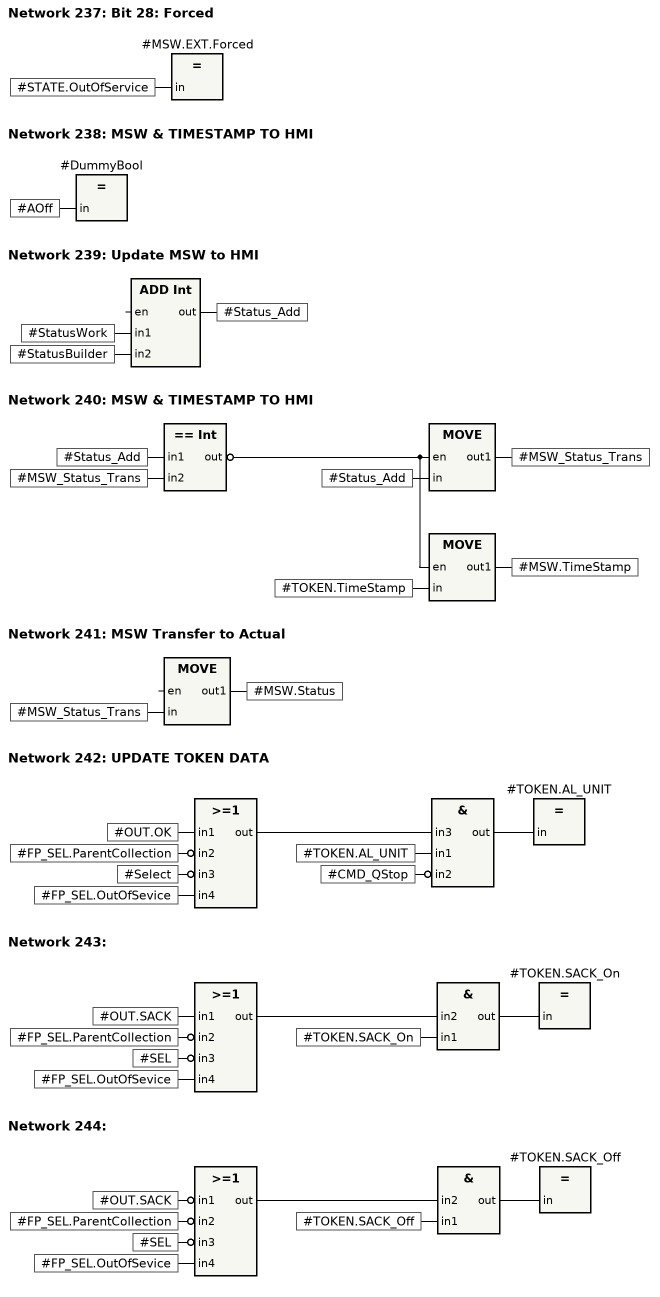
   #MSW.EXT.Forced := #STATE.OutOfService;
END_REGION

REGION Network 238: MSW & TIMESTAMP TO HMI
   #DummyBool := #AOff;
END_REGION

REGION Network 239: Update MSW to HMI
   #Status_Add := #StatusWork + #StatusBuilder;
END_REGION

REGION Network 240: MSW & TIMESTAMP TO HMI
   #_w1 := NOT (#Status_Add = #MSW_Status_Trans);
   IF #_w1 THEN
       #MSW_Status_Trans := #Status_Add;
       #MSW.TimeStamp := #TOKEN.TimeStamp;
   END_IF;
END_REGION

REGION Network 241: MSW Transfer to Actual
   #MSW.Status := #MSW_Status_Trans;
END_REGION

REGION Network 242: UPDATE TOKEN DATA
   #TOKEN.AL_UNIT := (#OUT.OK OR NOT #FP_SEL.ParentCollection OR NOT #Select OR #FP_SEL.OutOfSevice) AND #TOKEN.AL_UNIT AND NOT #CMD_QStop;
END_REGION

REGION Network 243
   // Build 005 - 24.June.2020 (MIA-US): Replace "Select" with "SEL"
   #TOKEN.SACK_On := (#OUT.SACK OR NOT #FP_SEL.ParentCollection OR NOT #SEL OR #FP_SEL.OutOfSevice) AND #TOKEN.SACK_On;
END_REGION

REGION Network 244
   #TOKEN.SACK_Off := (NOT #OUT.SACK OR NOT #FP_SEL.ParentCollection OR NOT #SEL OR #FP_SEL.OutOfSevice) AND #TOKEN.SACK_Off;
END_REGION

REGION Network 245
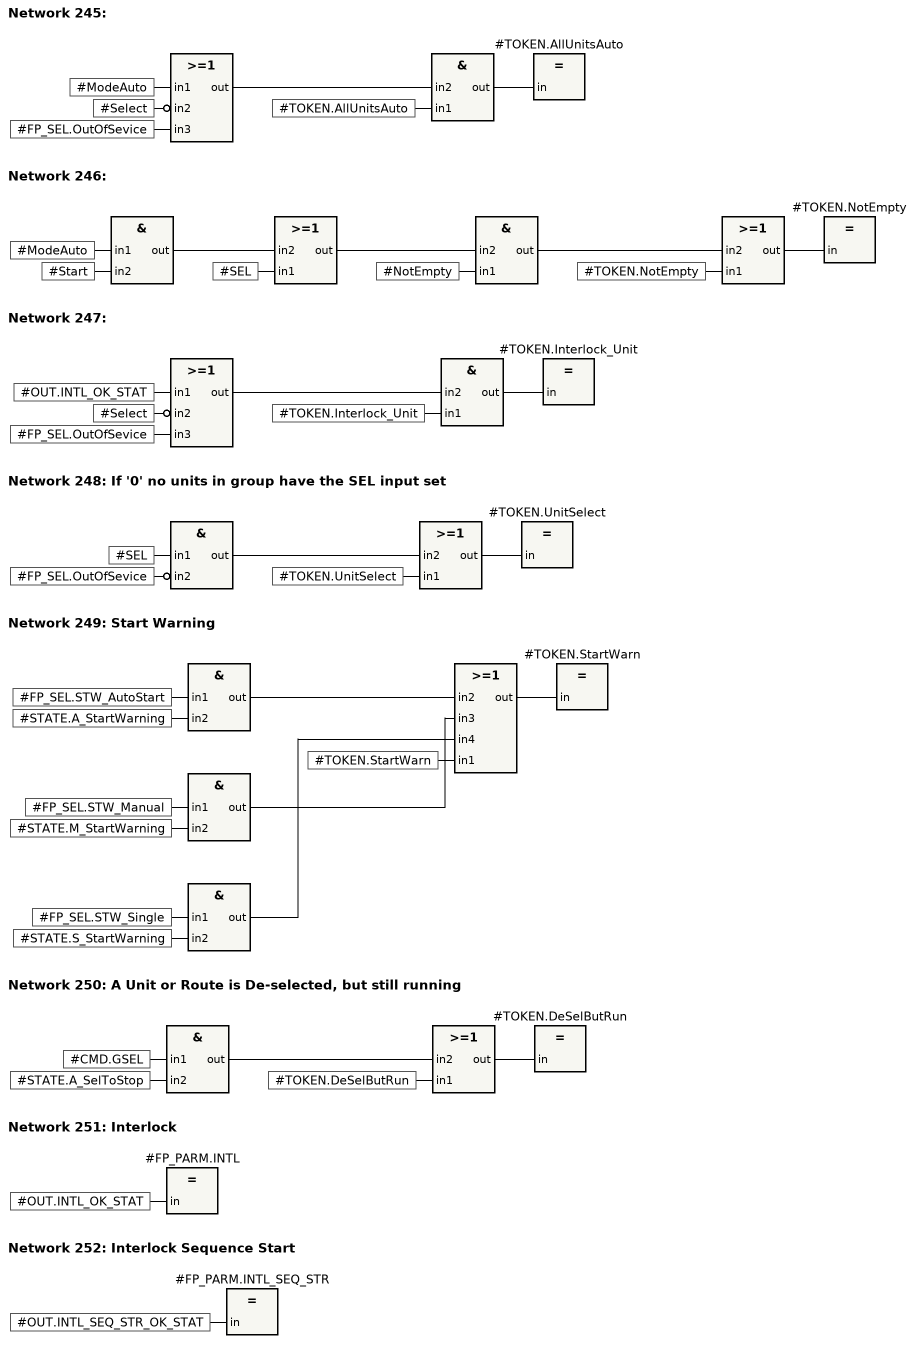
   #TOKEN.AllUnitsAuto := (#ModeAuto OR NOT #Select OR #FP_SEL.OutOfSevice) AND #TOKEN.AllUnitsAuto;
END_REGION

REGION Network 246
   #TOKEN.NotEmpty := (((#ModeAuto AND #Start) OR #SEL) AND #NotEmpty) OR #TOKEN.NotEmpty;
END_REGION

REGION Network 247
   #TOKEN.Interlock_Unit := (#OUT.INTL_OK_STAT OR NOT #Select OR #FP_SEL.OutOfSevice) AND #TOKEN.Interlock_Unit;
END_REGION

REGION Network 248: If '0' no units in group have the SEL input set
   #TOKEN.UnitSelect := (#SEL AND NOT #FP_SEL.OutOfSevice) OR #TOKEN.UnitSelect;
END_REGION

REGION Network 249: Start Warning
   #TOKEN.StartWarn := (#FP_SEL.STW_AutoStart AND #STATE.A_StartWarning) OR (#FP_SEL.STW_Manual AND #STATE.M_StartWarning) OR (#FP_SEL.STW_Single AND #STATE.S_StartWarning) OR #TOKEN.StartWarn;
END_REGION

REGION Network 250: A Unit or Route is De-selected, but still running
   #TOKEN.DeSelButRun := (#CMD.GSEL AND #STATE.A_SelToStop) OR #TOKEN.DeSelButRun;
END_REGION

REGION Network 251: Interlock
   #FP_PARM.INTL := #OUT.INTL_OK_STAT;
END_REGION

REGION Network 252: Interlock Sequence Start
   #FP_PARM.INTL_SEQ_STR := #OUT.INTL_SEQ_STR_OK_STAT;
END_REGION

REGION Network 253: Interlock Status to HMI
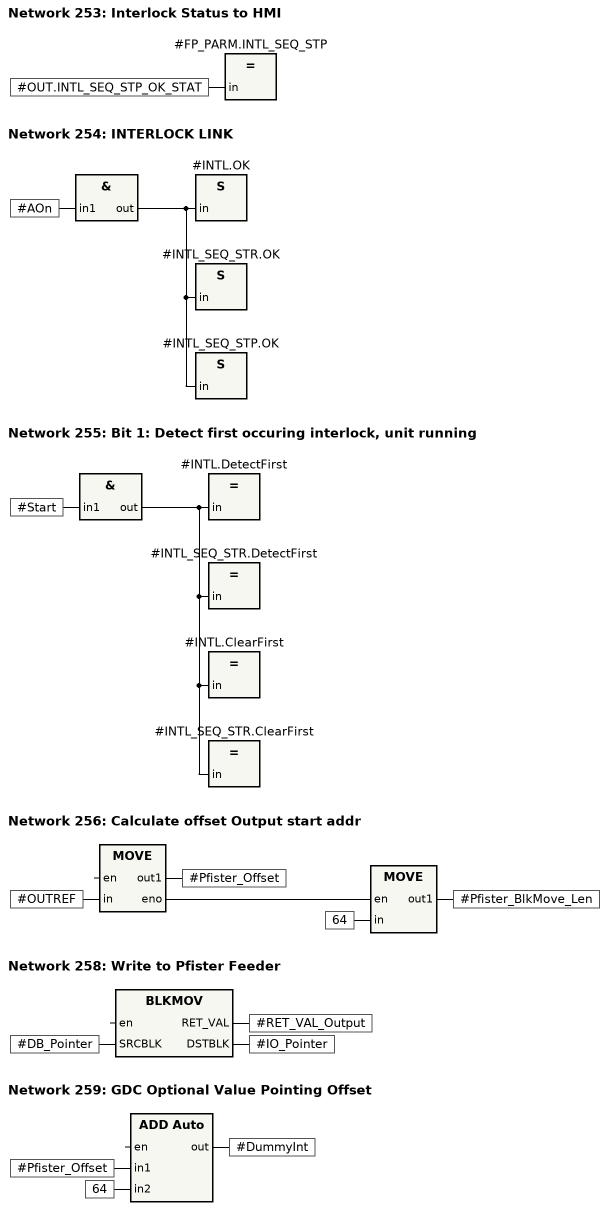
   #FP_PARM.INTL_SEQ_STP := #OUT.INTL_SEQ_STP_OK_STAT;
END_REGION

REGION Network 254: INTERLOCK LINK
   IF #AOn THEN
       #INTL.OK := TRUE;
       #INTL_SEQ_STR.OK := TRUE;
       #INTL_SEQ_STP.OK := TRUE;
   END_IF;
END_REGION

REGION Network 255: Bit 1: Detect first occuring interlock, unit running
   #INTL.DetectFirst := #Start;
   #INTL_SEQ_STR.DetectFirst := #Start;
   #INTL.ClearFirst := #Start;
   #INTL_SEQ_STR.ClearFirst := #Start;
END_REGION

REGION Network 256: Calculate offset Output start addr
   #Pfister_Offset := #OUTREF;
   #Pfister_BlkMove_Len := 64;
END_REGION

REGION Network 257 (STL): Target Pointers Sending Output Data
         LAR1;  // Make AR1 pointer to Unit Output
         L     16#10;  // ANY Syntax ID
         T     LB[AR1, P#0.0];  // ..Store Byte 0
         L     16#02;  // Data Type = Byte
         T     LB[AR1, P#1.0];  // ..Store Byte 1
         L     #Pfister_BlkMove_Len;  // Load Packed length
         T     LW[AR1, P#2.0];  // ..Store byte 2/3
         L     0;  // used with DB else "0"
         T     LW[AR1, P#4.0];  // ..Store byte 4/5
         L     #Pfister_Offset;  // Source offset (Variable for Node's)
         SLD   3;  // with offset
         OD    16#8200_0000;  // Output Area (I/O) Code (S7)
         T     LD[AR1, P#6.0];  // ..Store byte 6/7/8/9

         LAR1;  // Load start point of cyclic data
         TAR1  #DummyDWord;  // Store in temp. point
         L     #DummyDWord;  // Load temp. point
         T     #Addr_InstanceDB;  // Store start point as DB address

         LAR1;  // Make AR1 point to calling program stack
         L     16#10;  // ANY Syntax ID
         T     LB[AR1, P#0.0];  // ..Store Byte 0
         L     16#02;  // Data Type = Byte
         T     LB[AR1, P#1.0];  // ..Store Byte 1
         L     #Pfister_BlkMove_Len;  // Load Packed length
         T     LW[AR1, P#2.0];  // ..Store Byte 2/3
         L     #BlockInfo.DB_Number;  // used with DB use No. else "0"
         T     LW[AR1, P#4.0];  // ..Store byte 4/5
         L     #Addr_InstanceDB;  // Load Instance DB Start address
         L     16#8500_0000;
         -D;
         L     16#8400_0000;
         +D;
         T     LD[AR1, P#6.0];  // ..Store byte 6/7/8/9
END_REGION

REGION Network 258: Write to Pfister Feeder
   #RET_VAL_Output := BLKMOV(SRCBLK := #DB_Pointer, DSTBLK => #IO_Pointer);
END_REGION

REGION Network 259: GDC Optional Value Pointing Offset
   // Build 07 - 09 Jan 2022(VIV-IN) GDC Controller Function Type Added
   #DummyInt := #Pfister_Offset + 64;
END_REGION

REGION Network 260 (STL): Target Pointers Sending GDC Output Data
   // Build 07 - 09 Jan 2022(VIV-IN) GDC Controller Function Type Added
         LAR1;  // Make AR1 pointer to Unit Output
         L     B#16#10;  // ANY Syntax ID
         T     LB [AR1,P#0.0];  // ..Store Byte 0
         L     B#16#2;  // Data Type = Byte
         T     LB [AR1,P#1.0];  // ..Store Byte 1
         L     8;  // Load Packed length
         T     LW [AR1,P#2.0];  // ..Store byte 2/3
         L     0;  // used with DB else "0"
         T     LW [AR1,P#4.0];  // ..Store byte 4/5
         L     #DummyInt;  // Source offset (Variable for Node's)
         SLD   3;  // with offset
         OD    DW#16#82000000;  // Output Area (I/O) Code (S7)
         T     LD [AR1,P#6.0];  // ..Store byte 6/7/8/9
END_REGION

REGION Network 261: GDC Optional Read Value Write Byte 0 & 1
   // Build 07 - 09 Jan 2022(VIV-IN) GDC Controller Function Type Added
   // Build 017 - 09 Jan 2022 [viv-in] : GDC Controller Function Type Added
   // GDC Controller Optinal Read Value
   // 
   // 19 - Feeder Configuration
   // 20 - Firmware
   // 21- Range Feed
   // 22 - Range Pre Hopper
   // 13 - Total OLC
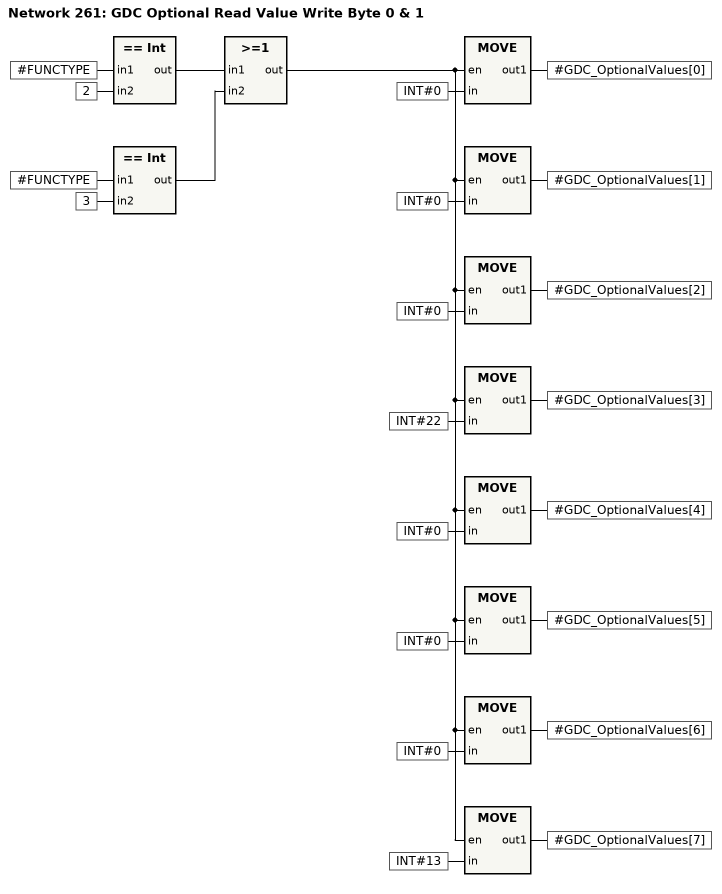
   IF (#FUNCTYPE = 2) OR (#FUNCTYPE = 3) THEN
       #GDC_OptionalValues[0] := INT#0;
       #GDC_OptionalValues[1] := INT#0;
       #GDC_OptionalValues[2] := INT#0;
       #GDC_OptionalValues[3] := INT#22;
       #GDC_OptionalValues[4] := INT#0;
       #GDC_OptionalValues[5] := INT#0;
       #GDC_OptionalValues[6] := INT#0;
       #GDC_OptionalValues[7] := INT#13;
   END_IF;
END_REGION

REGION Network 262: FDC Select - Write "0"
   // Build 07 - 09 Jan 2022(VIV-IN) GDC Controller Function Type Added
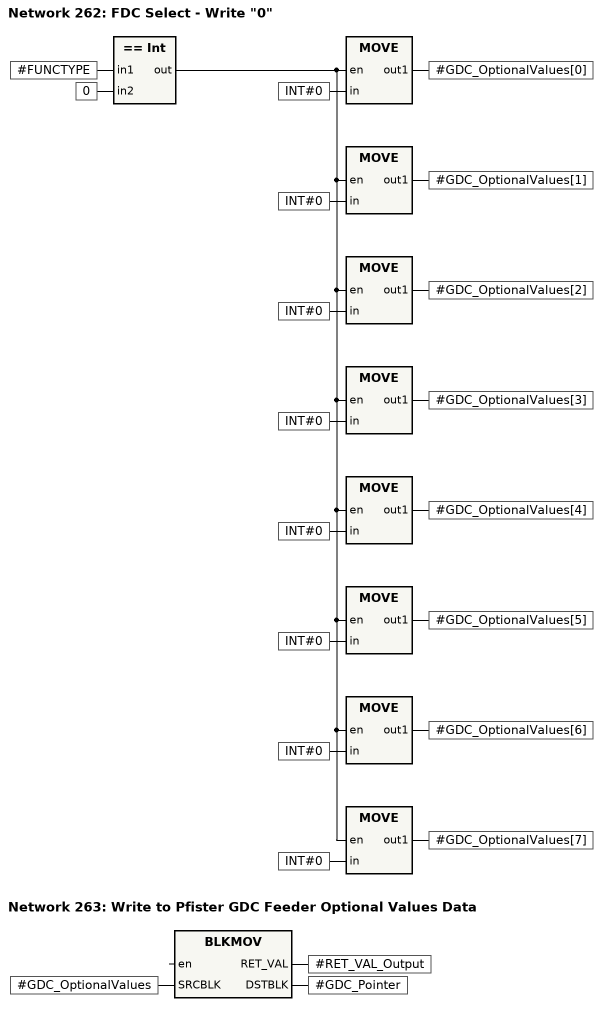
   IF #FUNCTYPE = 0 THEN
       #GDC_OptionalValues[0] := INT#0;
       #GDC_OptionalValues[1] := INT#0;
       #GDC_OptionalValues[2] := INT#0;
       #GDC_OptionalValues[3] := INT#0;
       #GDC_OptionalValues[4] := INT#0;
       #GDC_OptionalValues[5] := INT#0;
       #GDC_OptionalValues[6] := INT#0;
       #GDC_OptionalValues[7] := INT#0;
   END_IF;
END_REGION

REGION Network 263: Write to Pfister GDC Feeder Optional Values Data
   // Build 07 - 09 Jan 2022(VIV-IN) GDC Controller Function Type Added
   #RET_VAL_Output := BLKMOV(SRCBLK := #GDC_OptionalValues, DSTBLK => #GDC_Pointer);
END_REGION

REGION Network 264: GDC Firmware Read
   // Build 07 - 09 Jan 2022(VIV-IN) GDC Controller Function Type Added
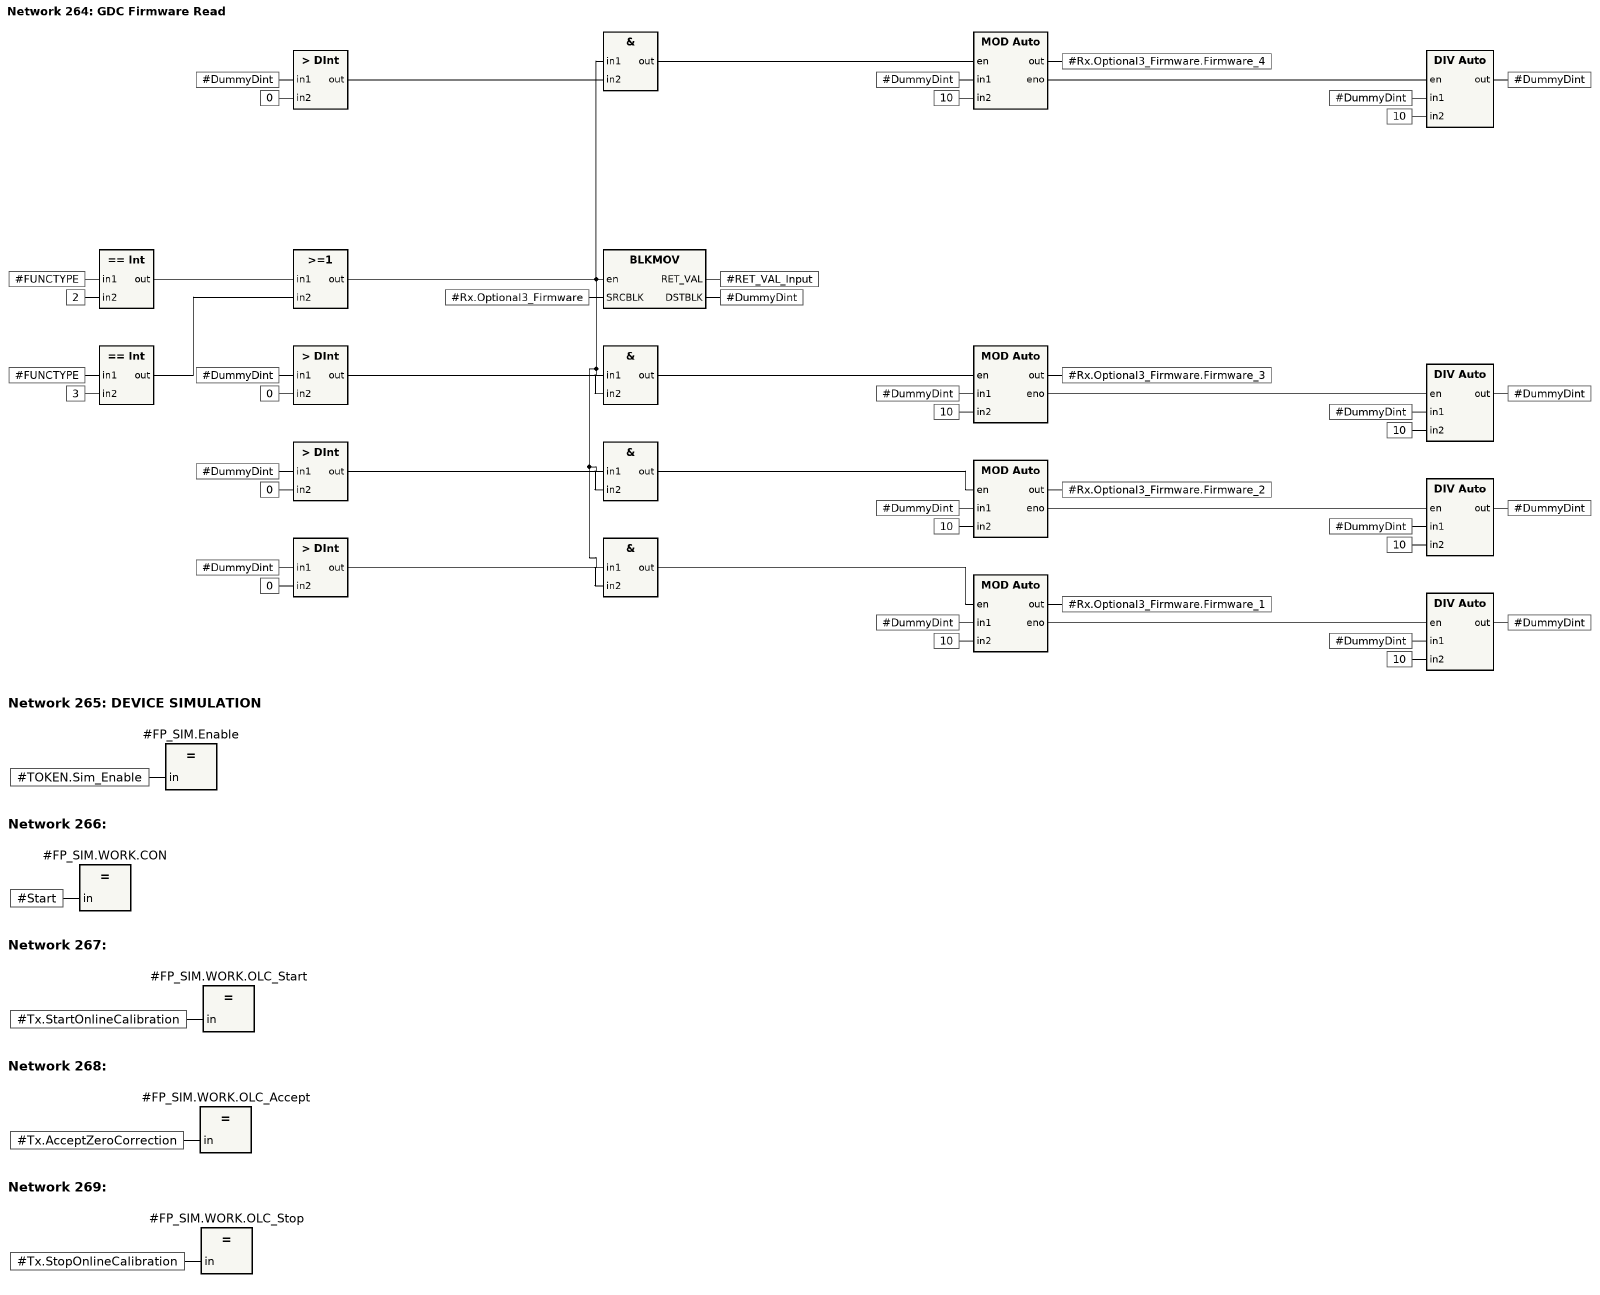
   #_w1 := (#FUNCTYPE = 2) OR (#FUNCTYPE = 3);
   IF #_w1 THEN #RET_VAL_Input := BLKMOV(SRCBLK := #Rx.Optional3_Firmware, DSTBLK => #DummyDint); END_IF;
   IF #_w1 AND (#DummyDint > 0) THEN
       #Rx.Optional3_Firmware.Firmware_4 := #DummyDint MOD 10;
       #DummyDint := #DummyDint / 10;
   END_IF;
   IF #_w1 AND (#DummyDint > 0) THEN
       #Rx.Optional3_Firmware.Firmware_3 := #DummyDint MOD 10;
       #DummyDint := #DummyDint / 10;
   END_IF;
   IF #_w1 AND (#DummyDint > 0) THEN
       #Rx.Optional3_Firmware.Firmware_2 := #DummyDint MOD 10;
       #DummyDint := #DummyDint / 10;
   END_IF;
   IF #_w1 AND (#DummyDint > 0) THEN
       #Rx.Optional3_Firmware.Firmware_1 := #DummyDint MOD 10;
       #DummyDint := #DummyDint / 10;
   END_IF;
END_REGION

REGION Network 265: DEVICE SIMULATION
   #FP_SIM.Enable := #TOKEN.Sim_Enable;
END_REGION

REGION Network 266
   #FP_SIM.WORK.CON := #Start;
END_REGION

REGION Network 267
   #FP_SIM.WORK.OLC_Start := #Tx.StartOnlineCalibration;
END_REGION

REGION Network 268
   #FP_SIM.WORK.OLC_Accept := #Tx.AcceptZeroCorrection;
END_REGION

REGION Network 269
   #FP_SIM.WORK.OLC_Stop := #Tx.StopOnlineCalibration;
END_REGION

REGION Network 270
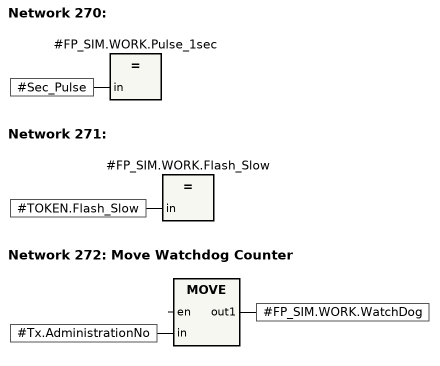
   #FP_SIM.WORK.Pulse_1sec := #Sec_Pulse;
END_REGION

REGION Network 271
   #FP_SIM.WORK.Flash_Slow := #TOKEN.Flash_Slow;
END_REGION

REGION Network 272: Move Watchdog Counter
   #FP_SIM.WORK.WatchDog := #Tx.AdministrationNo;
END_REGION

REGION Network 273: Write STAT to OUT
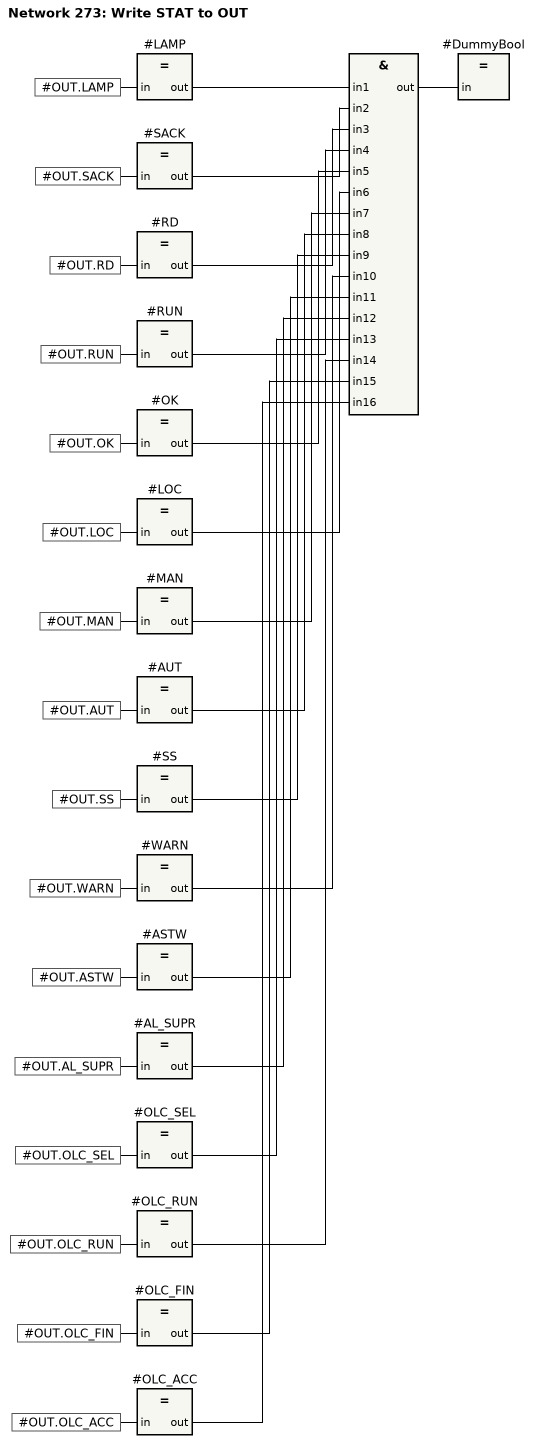
   #LAMP := #OUT.LAMP;
   #SACK := #OUT.SACK;
   #RD := #OUT.RD;
   #RUN := #OUT.RUN;
   #OK := #OUT.OK;
   #LOC := #OUT.LOC;
   #MAN := #OUT.MAN;
   #AUT := #OUT.AUT;
   #SS := #OUT.SS;
   #WARN := #OUT.WARN;
   #ASTW := #OUT.ASTW;
   #AL_SUPR := #OUT.AL_SUPR;
   #OLC_SEL := #OUT.OLC_SEL;
   #OLC_RUN := #OUT.OLC_RUN;
   #OLC_FIN := #OUT.OLC_FIN;
   #OLC_ACC := #OUT.OLC_ACC;
   #DummyBool := #OUT.LAMP AND #OUT.SACK AND #OUT.RD AND #OUT.RUN AND #OUT.OK AND #OUT.LOC AND #OUT.MAN AND #OUT.AUT AND #OUT.SS AND #OUT.WARN AND #OUT.ASTW AND #OUT.AL_SUPR AND #OUT.OLC_SEL AND #OUT.OLC_RUN AND #OUT.OLC_FIN AND #OUT.OLC_ACC;
END_REGION
END_FUNCTION_BLOCK

FUNCTION_BLOCK "ACESYS_SPC"   // FB217, FBD
TITLE = ACESYS V8.0 - Build 007 - SPC Filter
{ S7_Optimized_Access := 'FALSE' }
AUTHOR : FLSmidth
FAMILY : ACESYS
NAME : SPC
VERSION : 8.0
   VAR_INPUT
      CMD : "ACESYS_GRP_CMD";
      INREF : Int;   // Main Input address
      OUTREF : Int;   // Main Output address
      NET : Int;   // Net number
      NODE : Int;   // Node Number
      FUNCTYPE : Int;   // Filter Types : 400, 800, 1691
      OPTIONS : Int;   // Filter Options: 1691 Options; 4= UniClean Filter, 8 = Fabri Clean Filter
      SEL : Bool := TRUE;   // Unit Select by User program
      ASTR : Bool := TRUE;   // Auto Start
      REM : Bool := TRUE;   // Unit in Remote operation
      ACK : Bool;   // Feedback from unit on alarm reset
      CO_SEC : Int;   // Enter number of compartments/Sections
      NO_AI : Int;   // Enter number of analog option card normally HE5910
      NO_DI : Int;   // Enter number of digital option card normally HE5910
      FCL : Bool;   // Forced Cleaning request
      PCL : Bool;   // Post Cleaning request
      CSTP : Bool;   // Stop Filter Valve cleaning stops but dampers continues until finish
   END_VAR
   VAR_OUTPUT
      INTL : "ACESYS_INTL";   // Interlock
      INTL_SEQ_STR : "ACESYS_INTL";   // Interlock Sequence Start
      INTL_SEQ_STP : "ACESYS_INTL";   // Interlock Sequence Stop
      LAMP : Bool;   // Lamp 1
      SACK : Bool;   // Start Acknowledge
      RD : Bool;   // Run delayed 1
      RUN : Bool;   // Run 1
      OK : Bool;   // Unit Status OK (no alarms)
      LOC : Bool;   // Unit in Local Mode
      MAN : Bool;   // Unit in Manual Mode
      AUT : Bool;   // Unit in Auto Mode
      SS : Bool;   // Unit in Single Start Mode
      RES : Bool;   // Reset to unit
      ASTW : Bool;   // Start warning
      AL_SUPR : Bool;   // Supress Child Alarms
      FRC_CL : Bool;   // Force Cleaning is selected
      PST_CL : Bool;   // Post Cleaning is selected
      LPA : Bool;   // Local Panel is Active
      RLC : Bool;   // Remote Keypad is disabled
      SFLT : Bool;   // SPC has problems on the profibus network
      DP : Real;   // Differential Pressure
      MSW : "ACESYS_HMI_STAT_32T";
   END_VAR
   VAR_IN_OUT
      TOKEN : "ACESYS_TOKEN";
   END_VAR
   VAR
      BlockInfo : Struct
         Ace_Version : Int;   // Acesys Block Version Number
         Ace_BuildNo : Int;   // Acesys Block Build Number
         SPC_Version : Int;   // Acesys Block Version Number
         SPC_BuildNo : Int;   // Acesys Block Build Number
         State_Act : Int;   // Actual State Number
         State_Prev : Int;   // Previous State Number
         DB_Number : Int;   // Block Instance DB Number
      END_STRUCT;
      FP_CMD : Struct   // Faceplate Commands
         QuickStop : Bool;
         Spare_09 : Bool;
         Spare_10 : Bool;
         Spare_11 : Bool;
         Spare_12 : Bool;
         Spare_13 : Bool;
         Spare_14 : Bool;
         AckAlarm : Bool;
         Auto : Bool;
         Manual : Bool;
         Local : Bool;
         Start : Bool;
         Spare_04 : Bool;
         Stop : Bool;
         Reset : Bool;
         Spare_07 : Bool;
      END_STRUCT;
      FP_SEL : Struct   // Faceplate Selections
         STW_AutoStart : Bool;   // Faceplate Start Warning in Auto Start mode
         STW_Manual : Bool;   // Faceplate Start Warning in Manual mode
         STW_Single : Bool;   // Faceplate Start Warning in Single Start mode
         ParentSupress : Bool;   // Enable Parent Supress of alarms
         ParentCollection : Bool;   // Enable Inching in Manual Mode
         INCH_Man : Bool;   // Enable Inching in Manual Mode
         INCH_Loc : Bool;   // Enable Inching in Local Mode
         OutOfSevice : Bool;   // Select Out of Service
         WarningDrive : Bool;   // 0 = Failure Drive / 1 = Warning Drive
         Spare14 : Bool;
         Spare13 : Bool;
         Spare12 : Bool;
         Spare11 : Bool;
         Spare10 : Bool;
         Spare9 : Bool;
         Spare8 : Bool;
         Spare7 : Bool;
         Spare6 : Bool;
         Spare5 : Bool;
         Spare4 : Bool;
         Spare3 : Bool;
         Spare2 : Bool;
         Spare1 : Bool;
      END_STRUCT;
      FP_EN : Struct
         Mode_Auto : Bool;
         Mode_Man : Bool;
         Mode_Loc : Bool;
         Spare13 : Bool;
         Mode_SS_Field : Bool;
         Mode_SS_FP : Bool;
         PB_QStop : Bool;
         Spare9 : Bool;
         Spare8 : Bool;
         Spare7 : Bool;
         Spare6 : Bool;
         Spare5 : Bool;
         Spare4 : Bool;
         Spare3 : Bool;
         Spare2 : Bool;
         Spare1 : Bool;
      END_STRUCT;
      FP_DIM : Struct   // Faceplate Dimmed Buttons
         Auto : Bool;
         Local : Bool;
         Manual : Bool;
         Start : Bool;
         Stop : Bool;
         QStop : Bool;
         Reset : Bool;
         Q20 : Bool;   // Dimout Test Function
         Q22 : Bool;   // Dimout Test Valve No
         Q23_0 : Bool;   // Dimout Inlet Damper 1
         Q23_1 : Bool;   // Dimout Inlet Damper 2
         Q23_2 : Bool;   // Dimout Outlet Damper 1
         Q23_3 : Bool;   // Dimout Outlet Damper 2
         Q23_4 : Bool;   // Dimout Open
         Q23_5 : Bool;   // Dimout Close
         Q23_6 : Bool;   // Dimout Lock Isolation valve
         Q23_7 : Bool;   // Dimout Send
         Spare9 : Bool;
         Spare8 : Bool;
         Spare7 : Bool;
         Spare6 : Bool;
         Spare5 : Bool;
         Spare4 : Bool;
         Spare3 : Bool;
         Spare2 : Bool;
         Spare1 : Bool;
      END_STRUCT;
      FP_SHOW : Struct   // Faceplate Show Buttons
         PB_Auto : Bool;
         PB_Local : Bool;
         PB_Manual : Bool;
         PB_Start : Bool;
         PB_Stop : Bool;
         PB_QStop : Bool;
         ACK : Bool;
         REM : Bool;
         PB_Reset : Bool;
         ASTR : Bool;
         Spare04 : Bool;
         Spare03 : Bool;
         Spare02 : Bool;
         Spare01 : Bool;
      END_STRUCT;
      FP_PARM : Struct   // Faceplate Parameters
         StartWarn_Pre : Int;
         StartWarn_Acc : Int;
         RunDelay_Pre : Int;
         RunDelay_Acc : Int;
         DelayStart_Pre : Int;
         DelayStart_Acc : Int;
         DelayStop_Pre : Int;
         DelayStop_Acc : Int;
         ReturnMon_Pre : Int;
         ReturnMon_Acc : Int;
         StopReason : Int;
         INTL : Bool;   // Interlock
         INTL_SEQ_STR : Bool;   // Interlock Sequence Start
         INTL_SEQ_STP : Bool;   // Interlock Sequence Stop
         Spare12 : Bool;
         Spare11 : Bool;
         Spare10 : Bool;
         Spare09 : Bool;
         Spare08 : Bool;
         Spare07 : Bool;
         Spare06 : Bool;
         Spare05 : Bool;
         Spare04 : Bool;
         Spare03 : Bool;
         Spare02 : Bool;
         Spare01 : Bool;
      END_STRUCT;
      FP_SIM : "ACESYS_SIM_SPC";
      VolumeFlow : Int;   // Volume flow for SPC820
      RAnalogArray : Array[0..19] of Real;
      MemoryPool_cmd_ECS : Struct   // Command from ECS faceplates
         xFilterStart : Bool;
         xFilterStop : Bool;
         xEmergencyStop : Bool;
         xAlarmReset : Bool;
         xOfflineCleaning : Bool;
         xPostCleaning : Bool;
         xForcedCleaning : Bool;
         xSemiOfflineCleaning : Bool;
         LocalControlDisable : Bool;
         RemoteControl : Bool;
         OverwriteComp : Bool;
         x1691EVOMode : Bool;
         xDoublePurgeClean : Bool;
         xDoublePurgeCleanCCR : Bool;
         xCommandDummy1_6 : Bool;
         xCommandDummy1_7 : Bool;
         xCloseC1 : Bool;
         xCloseC2 : Bool;
         xCloseC3 : Bool;
         xCloseC4 : Bool;
         xCloseC5 : Bool;
         xCloseC6 : Bool;
         xCloseC7 : Bool;
         xCloseC8 : Bool;
         xCloseC9 : Bool;
         xCloseC10 : Bool;
         xCloseC11 : Bool;
         xCloseC12 : Bool;
         xCloseC13 : Bool;
         xCloseC14 : Bool;
         xCloseC15 : Bool;
         xCloseC16 : Bool;
         xCloseC17 : Bool;
         xCloseC18 : Bool;
         xCloseC19 : Bool;
         xCloseC20 : Bool;
         xCloseC21 : Bool;
         xCloseC22 : Bool;
         xCloseC23 : Bool;
         xCloseC24 : Bool;
         xCleanC1 : Bool;
         xCleanC2 : Bool;
         xCleanC3 : Bool;
         xCleanC4 : Bool;
         xCleanC5 : Bool;
         xCleanC6 : Bool;
         xCleanC7 : Bool;
         xCleanC8 : Bool;
         xCleanC9 : Bool;
         xCleanC10 : Bool;
         xCleanC11 : Bool;
         xCleanC12 : Bool;
         xCleanC13 : Bool;
         xCleanC14 : Bool;
         xCleanC15 : Bool;
         xCleanC16 : Bool;
         xCleanC17 : Bool;
         xCleanC18 : Bool;
         xCleanC19 : Bool;
         xCleanC20 : Bool;
         xCleanC21 : Bool;
         xCleanC22 : Bool;
         xCleanC23 : Bool;
         xCleanC24 : Bool;
         xDELTAP_lower_Offset : Int;
         xDELTAP_higher_Offset : Int;
         xEXTRA_Pause1 : Int;
         xEXTRA_Pause2 : Int;
         xReserved16 : Byte;
         xReserved17 : Byte;
         xReserved18 : Byte;
         xReserved19 : Byte;
         xTestCommandValue : Byte;
         xTestCompartmentNo : Byte;
         xTestValveNo : Byte;
         xTestInletDamper1 : Bool;
         xTestInletDamper2 : Bool;
         xTestOutletDamper1 : Bool;
         xTestOutletDamper2 : Bool;
         xTestDamperOpen : Bool;
         xTestDamperClose : Bool;
         xUnlockIsolationValve : Bool;
         xTestSend : Bool;
         xReserved24 : Byte;
         xReserved25 : Byte;
         xReserved26 : Byte;
         xReserved27 : Byte;
         xReserved28 : Byte;
         xReserved29 : Byte;
         CompartmentInfoNo : Byte;
         C1_CLS : Bool;
         C2_CLS : Bool;
         C3_CLS : Bool;
         C4_CLS : Bool;
         C5_CLS : Bool;
         C6_CLS : Bool;
         C7_CLS : Bool;
         C8_CLS : Bool;
         C9_CLS : Bool;
         C10_CLS : Bool;
         C11_CLS : Bool;
         C12_CLS : Bool;
         C13_CLS : Bool;
         C14_CLS : Bool;
         C15_CLS : Bool;
         C16_CLS : Bool;
         C17_CLS : Bool;
         C18_CLS : Bool;
         C19_CLS : Bool;
         C20_CLS : Bool;
         C21_CLS : Bool;
         C22_CLS : Bool;
         C23_CLS : Bool;
         C24_CLS : Bool;
      END_STRUCT;
      MemoryPool_Status : Struct   // Status to ECS faceplates
         STATUS : Struct
            IW00_0 : Bool;   // Cleaning activated
            IW00_1 : Bool;   // Filter stopped (Emergency)
            IW00_2 : Bool;   // Off-line cleaning activated
            IW00_3 : Bool;   // Cleaning cycle in operation
            IW00_4 : Bool;   // After cleaning in operation
            IW00_5 : Bool;   // Force cleaning in operation
            IW00_6 : Bool;   // Compartment cleaning in operation
            IW00_7 : Bool;   // Local Control activated
            IW01_0 : Bool;   // Test actived
            IW01_1 : Bool;   // Reserved
            IW01_2 : Bool;   // Reserved
            IW01_3 : Bool;   // Semi Offline Cleaning Status
            IW01_4 : Bool;   // Double Purge Cleaning Status
            IW01_5 : Bool;   // Reserved
            IW01_6 : Bool;   // Reserved
            IW01_7 : Bool;   // Reserved
            IB02 : Byte;   // Actual Compartment
            IB03 : Byte;   // Actual valve
            IW04_0 : Bool;   // Compartment 1 Closed
            IW04_1 : Bool;   // Compartment 2 Closed
            IW04_2 : Bool;   // Compartment 3 Closed
            IW04_3 : Bool;   // Compartment 4 Closed
            IW04_4 : Bool;   // Compartment 5 Closed
            IW04_5 : Bool;   // Compartment 6 Closed
            IW04_6 : Bool;   // Compartment 7 Closed
            IW04_7 : Bool;   // Compartment 8 Closed
            IW05_0 : Bool;   // Compartment 9 Closed
            IW05_1 : Bool;   // Compartment 10 Closed
            IW05_2 : Bool;   // Compartment 11 Closed
            IW05_3 : Bool;   // Compartment 12 Closed
            IW05_4 : Bool;   // Compartment 13 Closed
            IW05_5 : Bool;   // Compartment 14 Closed
            IW05_6 : Bool;   // Compartment 15 Closed
            IW05_7 : Bool;   // Compartment 16 Closed
            IW06_0 : Bool;   // Compartment 17 Closed
            IW06_1 : Bool;   // Compartment 18 Closed
            IW06_2 : Bool;   // Compartment 19 Closed
            IW06_3 : Bool;   // Compartment 20 Closed
            IW06_4 : Bool;   // Compartment 21 Closed
            IW06_5 : Bool;   // Compartment 22 Closed
            IW06_6 : Bool;   // Compartment 23 Closed
            IW06_7 : Bool;   // Compartment 24 Closed
            IW07_0 : Bool;   // Compartment 1 cleaning in operation
            IW07_1 : Bool;   // Compartment 2 cleaning in operation
            IW07_2 : Bool;   // Compartment 3 cleaning in operation
            IW07_3 : Bool;   // Compartment 4 cleaning in operation
            IW07_4 : Bool;   // Compartment 5 cleaning in operation
            IW07_5 : Bool;   // Compartment 6 cleaning in operation
            IW07_6 : Bool;   // Compartment 7 cleaning in operation
            IW07_7 : Bool;   // Compartment 8 cleaning in operation
            IW08_0 : Bool;   // Compartment 9 cleaning in operation
            IW08_1 : Bool;   // Compartment 10 cleaning in operation
            IW08_2 : Bool;   // Compartment 11 cleaning in operation
            IW08_3 : Bool;   // Compartment 12 cleaning in operation
            IW08_4 : Bool;   // Compartment 13 cleaning in operation
            IW08_5 : Bool;   // Compartment 14 cleaning in operation
            IW08_6 : Bool;   // Compartment 15 cleaning in operation
            IW08_7 : Bool;   // Compartment 16 cleaning in operation
            IW09_0 : Bool;   // Compartment 17 cleaning in operation
            IW09_1 : Bool;   // Compartment 18 cleaning in operation
            IW09_2 : Bool;   // Compartment 19 cleaning in operation
            IW09_3 : Bool;   // Compartment 20 cleaning in operation
            IW09_4 : Bool;   // Compartment 21 cleaning in operation
            IW09_5 : Bool;   // Compartment 22 cleaning in operation
            IW09_6 : Bool;   // Compartment 23 cleaning in operation
            IW09_7 : Bool;   // Compartment 24 cleaning in operation
            IW10_0 : Bool;   // General Alarm
            IW10_1 : Bool;   // Differential pressure alarm
            IW10_2 : Bool;   // Compressed air system fault
            IW10_3 : Bool;   // Manifold pressure alarm
            IW10_4 : Bool;   // Isolation valve malfunction
            IW10_5 : Bool;   // Valve malfunction
            IW10_6 : Bool;   // Hopper high level
            IW10_7 : Bool;   // Dust high level
            IW11_0 : Bool;   // Inlet damper alarm
            IW11_1 : Bool;   // Outlet damper alarm
            IW11_2 : Bool;   // CAN-Bus error
            IW11_3 : Bool;   // Reserved
            IW11_4 : Bool;   // Reserved
            IW11_5 : Bool;   // Reserved
            IW11_6 : Bool;   // Reserved
            IW11_7 : Bool;   // Reserved
            IW12_0 : Bool;   // Differential pressure 1. High level alarm
            IW12_1 : Bool;   // Differential pressure 2. High level alarm
            IW12_2 : Bool;   // Differential pressure Low level alarm
            IW12_3 : Bool;   // Differential pressure Sensor fault
            IW12_4 : Bool;   // System pressure High level alarm
            IW12_5 : Bool;   // System pressure Low level alarm
            IW12_6 : Bool;   // System pressure Sensor fault
            IW12_7 : Bool;   // Reserved
            IB13 : Byte;   // Reserved
            IB14 : Byte;   // Reserved
            IB15 : Byte;   // Reserved
            IB16 : Byte;   // Reserved
            IB17 : Byte;   // Reserved
            IB18 : Byte;   // Reserved
            IB19 : Byte;   // Reserved
         END_STRUCT;
         COMPARTMENT_VIEW : Array[0..3] of Byte;
         COMPARTMENT_VIEW_DIAG : Array[0..3] of Byte;
         SYSTEM_DIAG : Array[0..11] of Byte;
         DIAG_EXTRAANALOG : Array[0..4] of Byte;
      END_STRUCT;
      TYPE_800_DI : Array[0..3] of Byte;   // Possible Digital Card Arrangements
      ErrorCompartment1 : Bool;
      ErrorCompartment2 : Bool;
      ErrorCompartment3 : Bool;
      ErrorCompartment4 : Bool;
      ErrorCompartment5 : Bool;
      ErrorCompartment6 : Bool;
      ErrorCompartment7 : Bool;
      ErrorCompartment8 : Bool;
      ErrorCompartment9 : Bool;
      ErrorCompartment10 : Bool;
      ErrorCompartment11 : Bool;
      ErrorCompartment12 : Bool;
      ErrorCompartment13 : Bool;
      ErrorCompartment14 : Bool;
      ErrorCompartment15 : Bool;
      ErrorCompartment16 : Bool;
      ErrorCompartment17 : Bool;
      ErrorCompartment18 : Bool;
      ErrorCompartment19 : Bool;
      ErrorCompartment20 : Bool;
      ErrorCompartment21 : Bool;
      ErrorCompartment22 : Bool;
      ErrorCompartment23 : Bool;
      ErrorCompartment24 : Bool;
      ErrorCompart_Spare25 : Bool;
      ErrorCompart_Spare26 : Bool;
      ErrorCompart_Spare27 : Bool;
      ErrorCompart_Spare28 : Bool;
      ErrorCompart_Spare29 : Bool;
      ErrorCompart_Spare30 : Bool;
      ErrorCompart_Spare31 : Bool;
      ErrorCompart_Spare32 : Bool;
      TYPE_800_AI : Array[0..19] of Word;   // Possible Analog Card Arrangements
      TYPE_800_CHAMBERS : Array[0..95] of Byte;   // Possible Chamber arangements Max 24
      STATE : Struct
         A_AutoStart : Bool;
         A_DelayedStart : Bool;
         A_DelayedStop : Bool;
         A_Running : Bool;
         A_Selected : Bool;
         A_SelToStop : Bool;
         A_Stopping : Bool;
         A_SeqStart : Bool;
         A_SeqStop : Bool;
         A_Starting : Bool;
         A_StartWarning : Bool;
         A_Stopped : Bool;
         S_AutoStart : Bool;
         S_Running : Bool;
         S_Starting : Bool;
         S_StartWarning : Bool;
         S_Stopped : Bool;
         M_Running : Bool;
         M_Starting : Bool;
         M_StartWarning : Bool;
         M_Stopped : Bool;
         L_Running : Bool;
         L_Stopped : Bool;
         Alarm : Bool;
         Interlock : Bool;
         EmergencyStop : Bool;
         OutOfService : Bool;
      END_STRUCT;
      DiagnosticData : Struct
         DPDiagnostics : Struct
            StationStatus : Struct
               DPSlvNotFound : Bool;   // Station 1 Information
               DataExchangeNotReady : Bool;   // Station 1 Information
               ConfigDataIncorrect : Bool;   // Station 1 Information
               NewErrorAvailable : Bool;   // Station 1 Information
               FunctionNotAllowed : Bool;   // Station 1 Information
               DPReplyInvalid : Bool;   // Station 1 Information
               SoftwareConfigIncorrect : Bool;   // Station 1 Information
               DifferentConfigMaster : Bool;   // Station 1 Information
               SlvRequiresSetup : Bool;   // Station 2 Information
               SlvDiagnosticAvailable : Bool;   // Station 2 Information
               SlvSetThis : Bool;   // Station 2 Information
               ResponseMonitoringOn : Bool;   // Station 2 Information
               SlvReceivedFREEZE : Bool;   // Station 2 Information
               SlvreceivedSYNC : Bool;   // Station 2 Information
               Always0 : Bool;   // Station 2 Information
               SlvDeActivated : Bool;   // Station 2 Information
               NodeStatus3 : Byte;
               MASTER_PROFIBUS_ADDR : Byte;
               ManufactureCodeHiByte : Byte;
               ManufactureCodeLoByte : Byte;
            END_STRUCT;
            Ext_Header01 : Byte;
            InvalidParmaterData : Bool;
            InvalidConfiguration : Bool;
            InvalidCommand : Bool;
            InvalidTest : Bool;
            Ext_Header01_Reserved_04 : Bool;
            Ext_Header01_Reserved_05 : Bool;
            Ext_Header01_Reserved_06 : Bool;
            Ext_Header01_Reserved_07 : Bool;
            IO_Unit01_Disconnected : Bool;
            IO_Unit01_Malfunction : Bool;
            IO_Unit02_Disconnected : Bool;
            IO_Unit02_Malfunction : Bool;
            IO_Unit03_Disconnected : Bool;
            IO_Unit03_Malfunction : Bool;
            IO_Unit04_Disconnected : Bool;
            IO_Unit04_Malfunction : Bool;
            IO_Unit05_Disconnected : Bool;
            IO_Unit05_Malfunction : Bool;
            IO_Unit06_Disconnected : Bool;
            IO_Unit06_Malfunction : Bool;
            IO_Unit07_Disconnected : Bool;
            IO_Unit07_Malfunction : Bool;
            IO_Unit08_Disconnected : Bool;
            IO_Unit08_Malfunction : Bool;
            IO_Unit09_Disconnected : Bool;
            IO_Unit09_Malfunction : Bool;
            IO_Unit10_Disconnected : Bool;
            IO_Unit10_Malfunction : Bool;
            IO_Unit11_Disconnected : Bool;
            IO_Unit11_Malfunction : Bool;
            IO_Unit12_Disconnected : Bool;
            IO_Unit12_Malfunction : Bool;
            IO_State_Reserved_11 : Byte;
            IO_State_Reserved_12 : Byte;   // Not Used
            IO_State_Reserved_13 : Byte;   // Not Used
            IO_State_Reserved_14 : Byte;   // Not Used
            IO_State_Reserved_15 : Byte;   // Not Used
            IO_State_Reserved_16 : Byte;   // Not Used
            Header_Info_2 : Byte;   // Header 2
            C01_Slave01_Disconnected : Bool;
            C01_Slave01_Malfunction : Bool;
            C01_Slave02_Disconnected : Bool;
            C01_Slave02_Malfunction : Bool;
            C01_Reserved_4 : Bool;
            C01_Reserved_5 : Bool;
            C01_Reserved_6 : Bool;
            C01_Reserved_7 : Bool;
            C01_SenManifold_01_Break : Bool;
            C01_SenManifold_01_Short : Bool;
            C01_SenManifold_02_Break : Bool;
            C01_SenManifold_02_Short : Bool;
            C01_SenManifold_03_Break : Bool;
            C01_SenManifold_03_Short : Bool;
            C01_SenManifold_04_Break : Bool;
            C01_SenManifold_04_Short : Bool;
            C01_IsoVlvSlv_1_Break : Bool;
            C01_IsoVlvSlv_1_Short : Bool;
            C01_IsoVlvSlv_2_Break : Bool;
            C01_IsoVlvSlv_2_Short : Bool;
            C01_DustSensor_1_Break : Bool;
            C01_DustSensor_1_Short : Bool;
            C01_DustSensor_2_Break : Bool;
            C01_DustSensor_2_Short : Bool;
            C01_InDamper_1_NotOpn : Bool;
            C01_InDamper_1_NotCls : Bool;
            C01_InDamper_2_NotOpn : Bool;
            C01_InDamper_2_NotCls : Bool;
            C01_OutDamper_1_NotOpn : Bool;
            C01_OutDamper_1_NotCls : Bool;
            C01_OutDamper_2_NotOpn : Bool;
            C01_OutDamper_2_NotCls : Bool;
            C02_Slave01_Disconnected : Bool;
            C02_Slave01_Malfunction : Bool;
            C02_Slave02_Disconnected : Bool;
            C02_Slave02_Malfunction : Bool;
            C02_Reserved_4 : Bool;
            C02_Reserved_5 : Bool;
            C02_Reserved_6 : Bool;
            C02_SenManifold_01_Break : Bool;
            C02_Reserved_7 : Bool;
            C02_SenManifold_01_Short : Bool;
            C02_SenManifold_02_Break : Bool;
            C02_SenManifold_02_Short : Bool;
            C02_SenManifold_03_Break : Bool;
            C02_SenManifold_03_Short : Bool;
            C02_SenManifold_04_Break : Bool;
            C02_SenManifold_04_Short : Bool;
            C02_IsoVlvSlv_1_Break : Bool;
            C02_IsoVlvSlv_1_Short : Bool;
            C02_IsoVlvSlv_2_Break : Bool;
            C02_IsoVlvSlv_2_Short : Bool;
            C02_DustSensor_1_Break : Bool;
            C02_DustSensor_1_Short : Bool;
            C02_DustSensor_2_Break : Bool;
            C02_DustSensor_2_Short : Bool;
            C02_InDamper_1_NotOpn : Bool;
            C02_InDamper_1_NotCls : Bool;
            C02_InDamper_2_NotOpn : Bool;
            C02_InDamper_2_NotCls : Bool;
            C02_OutDamper_1_NotOpn : Bool;
            C02_OutDamper_1_NotCls : Bool;
            C02_OutDamper_2_NotOpn : Bool;
            C02_OutDamper_2_NotCls : Bool;
            C03_Slave01_Disconnected : Bool;
            C03_Slave01_Malfunction : Bool;
            C03_Slave02_Disconnected : Bool;
            C03_Slave02_Malfunction : Bool;
            C03_Reserved_4 : Bool;
            C03_Reserved_5 : Bool;
            C03_Reserved_6 : Bool;
            C03_Reserved_7 : Bool;
            C03_SenManifold_01_Break : Bool;
            C03_SenManifold_01_Short : Bool;
            C03_SenManifold_02_Break : Bool;
            C03_SenManifold_02_Short : Bool;
            C03_SenManifold_03_Break : Bool;
            C03_SenManifold_03_Short : Bool;
            C03_SenManifold_04_Break : Bool;
            C03_SenManifold_04_Short : Bool;
            C03_IsoVlvSlv_1_Break : Bool;
            C03_IsoVlvSlv_1_Short : Bool;
            C03_IsoVlvSlv_2_Break : Bool;
            C03_IsoVlvSlv_2_Short : Bool;
            C03_DustSensor_1_Break : Bool;
            C03_DustSensor_1_Short : Bool;
            C03_DustSensor_2_Break : Bool;
            C03_DustSensor_2_Short : Bool;
            C03_InDamper_1_NotOpn : Bool;
            C03_InDamper_1_NotCls : Bool;
            C03_InDamper_2_NotOpn : Bool;
            C03_InDamper_2_NotCls : Bool;
            C03_OutDamper_1_NotOpn : Bool;
            C03_OutDamper_1_NotCls : Bool;
            C03_OutDamper_2_NotOpn : Bool;
            C03_OutDamper_2_NotCls : Bool;
            C04_Slave01_Disconnected : Bool;
            C04_Slave01_Malfunction : Bool;
            C04_Slave02_Disconnected : Bool;
            C04_Slave02_Malfunction : Bool;
            C04_Reserved_4 : Bool;
            C04_Reserved_5 : Bool;
            C04_Reserved_6 : Bool;
            C04_Reserved_7 : Bool;
            C04_SenManifold_01_Break : Bool;
            C04_SenManifold_01_Short : Bool;
            C04_SenManifold_02_Break : Bool;
            C04_SenManifold_02_Short : Bool;
            C04_SenManifold_03_Break : Bool;
            C04_SenManifold_03_Short : Bool;
            C04_SenManifold_04_Break : Bool;
            C04_SenManifold_04_Short : Bool;
            C04_IsoVlvSlv_1_Break : Bool;
            C04_IsoVlvSlv_1_Short : Bool;
            C04_IsoVlvSlv_2_Break : Bool;
            C04_IsoVlvSlv_2_Short : Bool;
            C04_DustSensor_1_Break : Bool;
            C04_DustSensor_1_Short : Bool;
            C04_DustSensor_2_Break : Bool;
            C04_DustSensor_2_Short : Bool;
            C04_InDamper_1_NotOpn : Bool;
            C04_InDamper_1_NotCls : Bool;
            C04_InDamper_2_NotOpn : Bool;
            C04_InDamper_2_NotCls : Bool;
            C04_OutDamper_1_NotOpn : Bool;
            C04_OutDamper_1_NotCls : Bool;
            C04_OutDamper_2_NotOpn : Bool;
            C04_OutDamper_2_NotCls : Bool;
            C05_Slave01_Disconnected : Bool;
            C05_Slave01_Malfunction : Bool;
            C05_Slave02_Disconnected : Bool;
            C05_Slave02_Malfunction : Bool;
            C05_Reserved_4 : Bool;
            C05_Reserved_5 : Bool;
            C05_Reserved_6 : Bool;
            C05_Reserved_7 : Bool;
            C05_SenManifold_01_Break : Bool;
            C05_SenManifold_01_Short : Bool;
            C05_SenManifold_02_Break : Bool;
            C05_SenManifold_02_Short : Bool;
            C05_SenManifold_03_Break : Bool;
            C05_SenManifold_03_Short : Bool;
            C05_SenManifold_04_Break : Bool;
            C05_SenManifold_04_Short : Bool;
            C05_IsoVlvSlv_1_Break : Bool;
            C05_IsoVlvSlv_1_Short : Bool;
            C05_IsoVlvSlv_2_Break : Bool;
            C05_IsoVlvSlv_2_Short : Bool;
            C05_DustSensor_1_Break : Bool;
            C05_DustSensor_1_Short : Bool;
            C05_DustSensor_2_Break : Bool;
            C05_DustSensor_2_Short : Bool;
            C05_InDamper_1_NotOpn : Bool;
            C05_InDamper_1_NotCls : Bool;
            C05_InDamper_2_NotOpn : Bool;
            C05_InDamper_2_NotCls : Bool;
            C05_OutDamper_1_NotOpn : Bool;
            C05_OutDamper_1_NotCls : Bool;
            C05_OutDamper_2_NotOpn : Bool;
            C05_OutDamper_2_NotCls : Bool;
            C06_Slave01_Disconnected : Bool;
            C06_Slave01_Malfunction : Bool;
            C06_Slave02_Disconnected : Bool;
            C06_Slave02_Malfunction : Bool;
            C06_Reserved_4 : Bool;
            C06_Reserved_5 : Bool;
            C06_Reserved_6 : Bool;
            C06_Reserved_7 : Bool;
            C06_SenManifold_01_Break : Bool;
            C06_SenManifold_01_Short : Bool;
            C06_SenManifold_02_Break : Bool;
            C06_SenManifold_02_Short : Bool;
            C06_SenManifold_03_Break : Bool;
            C06_SenManifold_03_Short : Bool;
            C06_SenManifold_04_Break : Bool;
            C06_SenManifold_04_Short : Bool;
            C06_IsoVlvSlv_1_Break : Bool;
            C06_IsoVlvSlv_1_Short : Bool;
            C06_IsoVlvSlv_2_Break : Bool;
            C06_IsoVlvSlv_2_Short : Bool;
            C06_DustSensor_1_Break : Bool;
            C06_DustSensor_1_Short : Bool;
            C06_DustSensor_2_Break : Bool;
            C06_DustSensor_2_Short : Bool;
            C06_InDamper_1_NotOpn : Bool;
            C06_InDamper_1_NotCls : Bool;
            C06_InDamper_2_NotOpn : Bool;
            C06_InDamper_2_NotCls : Bool;
            C06_OutDamper_1_NotOpn : Bool;
            C06_OutDamper_1_NotCls : Bool;
            C06_OutDamper_2_NotOpn : Bool;
            C06_OutDamper_2_NotCls : Bool;
            C07_Slave01_Disconnected : Bool;
            C07_Slave01_Malfunction : Bool;
            C07_Slave02_Disconnected : Bool;
            C07_Slave02_Malfunction : Bool;
            C07_Reserved_4 : Bool;
            C07_Reserved_5 : Bool;
            C07_Reserved_6 : Bool;
            C07_Reserved_7 : Bool;
            C07_SenManifold_01_Break : Bool;
            C07_SenManifold_01_Short : Bool;
            C07_SenManifold_02_Break : Bool;
            C07_SenManifold_02_Short : Bool;
            C07_SenManifold_03_Break : Bool;
            C07_SenManifold_03_Short : Bool;
            C07_SenManifold_04_Break : Bool;
            C07_SenManifold_04_Short : Bool;
            C07_IsoVlvSlv_1_Break : Bool;
            C07_IsoVlvSlv_1_Short : Bool;
            C07_IsoVlvSlv_2_Break : Bool;
            C07_IsoVlvSlv_2_Short : Bool;
            C07_DustSensor_1_Break : Bool;
            C07_DustSensor_1_Short : Bool;
            C07_DustSensor_2_Break : Bool;
            C07_DustSensor_2_Short : Bool;
            C07_InDamper_1_NotOpn : Bool;
            C07_InDamper_1_NotCls : Bool;
            C07_InDamper_2_NotOpn : Bool;
            C07_InDamper_2_NotCls : Bool;
            C07_OutDamper_1_NotOpn : Bool;
            C07_OutDamper_1_NotCls : Bool;
            C07_OutDamper_2_NotOpn : Bool;
            C07_OutDamper_2_NotCls : Bool;
            C08_Slave01_Disconnected : Bool;
            C08_Slave01_Malfunction : Bool;
            C08_Slave02_Disconnected : Bool;
            C08_Slave02_Malfunction : Bool;
            C08_Reserved_4 : Bool;
            C08_Reserved_5 : Bool;
            C08_Reserved_6 : Bool;
            C08_Reserved_7 : Bool;
            C08_SenManifold_01_Break : Bool;
            C08_SenManifold_01_Short : Bool;
            C08_SenManifold_02_Break : Bool;
            C08_SenManifold_02_Short : Bool;
            C08_SenManifold_03_Break : Bool;
            C08_SenManifold_03_Short : Bool;
            C08_SenManifold_04_Break : Bool;
            C08_SenManifold_04_Short : Bool;
            C08_IsoVlvSlv_1_Break : Bool;
            C08_IsoVlvSlv_1_Short : Bool;
            C08_IsoVlvSlv_2_Break : Bool;
            C08_IsoVlvSlv_2_Short : Bool;
            C08_DustSensor_1_Break : Bool;
            C08_DustSensor_1_Short : Bool;
            C08_DustSensor_2_Break : Bool;
            C08_DustSensor_2_Short : Bool;
            C08_InDamper_1_NotOpn : Bool;
            C08_InDamper_1_NotCls : Bool;
            C08_InDamper_2_NotOpn : Bool;
            C08_InDamper_2_NotCls : Bool;
            C08_OutDamper_1_NotOpn : Bool;
            C08_OutDamper_1_NotCls : Bool;
            C08_OutDamper_2_NotOpn : Bool;
            C08_OutDamper_2_NotCls : Bool;
            Header_Info_3 : Byte;
            C09_Slave01_Disconnected : Bool;
            C09_Slave01_Malfunction : Bool;
            C09_Slave02_Disconnected : Bool;
            C09_Slave02_Malfunction : Bool;
            C09_Reserved_4 : Bool;
            C09_Reserved_5 : Bool;
            C09_Reserved_6 : Bool;
            C09_Reserved_7 : Bool;
            C09_SenManifold_01_Break : Bool;
            C09_SenManifold_01_Short : Bool;
            C09_SenManifold_02_Break : Bool;
            C09_SenManifold_02_Short : Bool;
            C09_SenManifold_03_Break : Bool;
            C09_SenManifold_03_Short : Bool;
            C09_SenManifold_04_Break : Bool;
            C09_SenManifold_04_Short : Bool;
            C09_IsoVlvSlv_1_Break : Bool;
            C09_IsoVlvSlv_1_Short : Bool;
            C09_IsoVlvSlv_2_Break : Bool;
            C09_IsoVlvSlv_2_Short : Bool;
            C09_DustSensor_1_Break : Bool;
            C09_DustSensor_1_Short : Bool;
            C09_DustSensor_2_Break : Bool;
            C09_DustSensor_2_Short : Bool;
            C09_InDamper_1_NotOpn : Bool;
            C09_InDamper_1_NotCls : Bool;
            C09_InDamper_2_NotOpn : Bool;
            C09_InDamper_2_NotCls : Bool;
            C09_OutDamper_1_NotOpn : Bool;
            C09_OutDamper_1_NotCls : Bool;
            C09_OutDamper_2_NotOpn : Bool;
            C09_OutDamper_2_NotCls : Bool;
            C10_Slave01_Disconnected : Bool;
            C10_Slave01_Malfunction : Bool;
            C10_Slave02_Disconnected : Bool;
            C10_Slave02_Malfunction : Bool;
            C10_Reserved_4 : Bool;
            C10_Reserved_5 : Bool;
            C10_Reserved_6 : Bool;
            C10_Reserved_7 : Bool;
            C10_SenManifold_01_Break : Bool;
            C10_SenManifold_01_Short : Bool;
            C10_SenManifold_02_Break : Bool;
            C10_SenManifold_02_Short : Bool;
            C10_SenManifold_03_Break : Bool;
            C10_SenManifold_03_Short : Bool;
            C10_SenManifold_04_Break : Bool;
            C10_SenManifold_04_Short : Bool;
            C10_IsoVlvSlv_1_Break : Bool;
            C10_IsoVlvSlv_1_Short : Bool;
            C10_IsoVlvSlv_2_Break : Bool;
            C10_IsoVlvSlv_2_Short : Bool;
            C10_DustSensor_1_Break : Bool;
            C10_DustSensor_1_Short : Bool;
            C10_DustSensor_2_Break : Bool;
            C10_DustSensor_2_Short : Bool;
            C10_InDamper_1_NotOpn : Bool;
            C10_InDamper_1_NotCls : Bool;
            C10_InDamper_2_NotOpn : Bool;
            C10_InDamper_2_NotCls : Bool;
            C10_OutDamper_1_NotOpn : Bool;
            C10_OutDamper_1_NotCls : Bool;
            C10_OutDamper_2_NotOpn : Bool;
            C10_OutDamper_2_NotCls : Bool;
            C11_Slave01_Disconnected : Bool;
            C11_Slave01_Malfunction : Bool;
            C11_Slave02_Disconnected : Bool;
            C11_Slave02_Malfunction : Bool;
            C11_Reserved_4 : Bool;
            C11_Reserved_5 : Bool;
            C11_Reserved_6 : Bool;
            C11_Reserved_7 : Bool;
            C11_SenManifold_01_Break : Bool;
            C11_SenManifold_01_Short : Bool;
            C11_SenManifold_02_Break : Bool;
            C11_SenManifold_02_Short : Bool;
            C11_SenManifold_03_Break : Bool;
            C11_SenManifold_03_Short : Bool;
            C11_SenManifold_04_Break : Bool;
            C11_SenManifold_04_Short : Bool;
            C11_IsoVlvSlv_1_Break : Bool;
            C11_IsoVlvSlv_1_Short : Bool;
            C11_IsoVlvSlv_2_Break : Bool;
            C11_IsoVlvSlv_2_Short : Bool;
            C11_DustSensor_1_Break : Bool;
            C11_DustSensor_1_Short : Bool;
            C11_DustSensor_2_Break : Bool;
            C11_DustSensor_2_Short : Bool;
            C11_InDamper_1_NotOpn : Bool;
            C11_InDamper_1_NotCls : Bool;
            C11_InDamper_2_NotOpn : Bool;
            C11_InDamper_2_NotCls : Bool;
            C11_OutDamper_1_NotOpn : Bool;
            C11_OutDamper_1_NotCls : Bool;
            C11_OutDamper_2_NotOpn : Bool;
            C11_OutDamper_2_NotCls : Bool;
            C12_Slave01_Disconnected : Bool;
            C12_Slave01_Malfunction : Bool;
            C12_Slave02_Disconnected : Bool;
            C12_Slave02_Malfunction : Bool;
            C12_Reserved_4 : Bool;
            C12_Reserved_5 : Bool;
            C12_Reserved_6 : Bool;
            C12_Reserved_7 : Bool;
            C12_SenManifold_01_Break : Bool;
            C12_SenManifold_01_Short : Bool;
            C12_SenManifold_02_Break : Bool;
            C12_SenManifold_02_Short : Bool;
            C12_SenManifold_03_Break : Bool;
            C12_SenManifold_03_Short : Bool;
            C12_SenManifold_04_Break : Bool;
            C12_SenManifold_04_Short : Bool;
            C12_IsoVlvSlv_1_Break : Bool;
            C12_IsoVlvSlv_1_Short : Bool;
            C12_IsoVlvSlv_2_Break : Bool;
            C12_IsoVlvSlv_2_Short : Bool;
            C12_DustSensor_1_Break : Bool;
            C12_DustSensor_1_Short : Bool;
            C12_DustSensor_2_Break : Bool;
            C12_DustSensor_2_Short : Bool;
            C12_InDamper_1_NotOpn : Bool;
            C12_InDamper_1_NotCls : Bool;
            C12_InDamper_2_NotOpn : Bool;
            C12_InDamper_2_NotCls : Bool;
            C12_OutDamper_1_NotOpn : Bool;
            C12_OutDamper_1_NotCls : Bool;
            C12_OutDamper_2_NotOpn : Bool;
            C12_OutDamper_2_NotCls : Bool;
            C13_Slave01_Disconnected : Bool;
            C13_Slave01_Malfunction : Bool;
            C13_Slave02_Disconnected : Bool;
            C13_Slave02_Malfunction : Bool;
            C13_Reserved_4 : Bool;
            C13_Reserved_5 : Bool;
            C13_Reserved_6 : Bool;
            C13_Reserved_7 : Bool;
            C13_SenManifold_01_Break : Bool;
            C13_SenManifold_01_Short : Bool;
            C13_SenManifold_02_Break : Bool;
            C13_SenManifold_02_Short : Bool;
            C13_SenManifold_03_Break : Bool;
            C13_SenManifold_03_Short : Bool;
            C13_SenManifold_04_Break : Bool;
            C13_SenManifold_04_Short : Bool;
            C13_IsoVlvSlv_1_Break : Bool;
            C13_IsoVlvSlv_1_Short : Bool;
            C13_IsoVlvSlv_2_Break : Bool;
            C13_IsoVlvSlv_2_Short : Bool;
            C13_DustSensor_1_Break : Bool;
            C13_DustSensor_1_Short : Bool;
            C13_DustSensor_2_Break : Bool;
            C13_DustSensor_2_Short : Bool;
            C13_InDamper_1_NotOpn : Bool;
            C13_InDamper_1_NotCls : Bool;
            C13_InDamper_2_NotOpn : Bool;
            C13_InDamper_2_NotCls : Bool;
            C13_OutDamper_1_NotOpn : Bool;
            C13_OutDamper_1_NotCls : Bool;
            C13_OutDamper_2_NotOpn : Bool;
            C13_OutDamper_2_NotCls : Bool;
            C14_Slave01_Disconnected : Bool;
            C14_Slave01_Malfunction : Bool;
            C14_Slave02_Disconnected : Bool;
            C14_Slave02_Malfunction : Bool;
            C14_Reserved_4 : Bool;
            C14_Reserved_5 : Bool;
            C14_Reserved_6 : Bool;
            C14_Reserved_7 : Bool;
            C14_SenManifold_01_Break : Bool;
            C14_SenManifold_01_Short : Bool;
            C14_SenManifold_02_Break : Bool;
            C14_SenManifold_02_Short : Bool;
            C14_SenManifold_03_Break : Bool;
            C14_SenManifold_03_Short : Bool;
            C14_SenManifold_04_Break : Bool;
            C14_SenManifold_04_Short : Bool;
            C14_IsoVlvSlv_1_Break : Bool;
            C14_IsoVlvSlv_1_Short : Bool;
            C14_IsoVlvSlv_2_Break : Bool;
            C14_IsoVlvSlv_2_Short : Bool;
            C14_DustSensor_1_Break : Bool;
            C14_DustSensor_1_Short : Bool;
            C14_DustSensor_2_Break : Bool;
            C14_DustSensor_2_Short : Bool;
            C14_InDamper_1_NotOpn : Bool;
            C14_InDamper_1_NotCls : Bool;
            C14_InDamper_2_NotOpn : Bool;
            C14_InDamper_2_NotCls : Bool;
            C14_OutDamper_1_NotOpn : Bool;
            C14_OutDamper_1_NotCls : Bool;
            C14_OutDamper_2_NotOpn : Bool;
            C14_OutDamper_2_NotCls : Bool;
            C15_Slave01_Disconnected : Bool;
            C15_Slave01_Malfunction : Bool;
            C15_Slave02_Disconnected : Bool;
            C15_Slave02_Malfunction : Bool;
            C15_Reserved_4 : Bool;
            C15_Reserved_5 : Bool;
            C15_Reserved_6 : Bool;
            C15_Reserved_7 : Bool;
            C15_SenManifold_01_Break : Bool;
            C15_SenManifold_01_Short : Bool;
            C15_SenManifold_02_Break : Bool;
            C15_SenManifold_02_Short : Bool;
            C15_SenManifold_03_Break : Bool;
            C15_SenManifold_03_Short : Bool;
            C15_SenManifold_04_Break : Bool;
            C15_SenManifold_04_Short : Bool;
            C15_IsoVlvSlv_1_Break : Bool;
            C15_IsoVlvSlv_1_Short : Bool;
            C15_IsoVlvSlv_2_Break : Bool;
            C15_IsoVlvSlv_2_Short : Bool;
            C15_DustSensor_1_Break : Bool;
            C15_DustSensor_1_Short : Bool;
            C15_DustSensor_2_Break : Bool;
            C15_DustSensor_2_Short : Bool;
            C15_InDamper_1_NotOpn : Bool;
            C15_InDamper_1_NotCls : Bool;
            C15_InDamper_2_NotOpn : Bool;
            C15_InDamper_2_NotCls : Bool;
            C15_OutDamper_1_NotOpn : Bool;
            C15_OutDamper_1_NotCls : Bool;
            C15_OutDamper_2_NotOpn : Bool;
            C15_OutDamper_2_NotCls : Bool;
            C16_Slave01_Disconnected : Bool;
            C16_Slave01_Malfunction : Bool;
            C16_Slave02_Disconnected : Bool;
            C16_Slave02_Malfunction : Bool;
            C16_Reserved_4 : Bool;
            C16_Reserved_5 : Bool;
            C16_Reserved_6 : Bool;
            C16_Reserved_7 : Bool;
            C16_SenManifold_01_Break : Bool;
            C16_SenManifold_01_Short : Bool;
            C16_SenManifold_02_Break : Bool;
            C16_SenManifold_02_Short : Bool;
            C16_SenManifold_03_Break : Bool;
            C16_SenManifold_03_Short : Bool;
            C16_SenManifold_04_Break : Bool;
            C16_SenManifold_04_Short : Bool;
            C16_IsoVlvSlv_1_Break : Bool;
            C16_IsoVlvSlv_1_Short : Bool;
            C16_IsoVlvSlv_2_Break : Bool;
            C16_IsoVlvSlv_2_Short : Bool;
            C16_DustSensor_1_Break : Bool;
            C16_DustSensor_1_Short : Bool;
            C16_DustSensor_2_Break : Bool;
            C16_DustSensor_2_Short : Bool;
            C16_InDamper_1_NotOpn : Bool;
            C16_InDamper_1_NotCls : Bool;
            C16_InDamper_2_NotOpn : Bool;
            C16_InDamper_2_NotCls : Bool;
            C16_OutDamper_1_NotOpn : Bool;
            C16_OutDamper_1_NotCls : Bool;
            C16_OutDamper_2_NotOpn : Bool;
            C16_OutDamper_2_NotCls : Bool;
            Header_Info_4 : Byte;
            C17_Slave01_Disconnected : Bool;
            C17_Slave01_Malfunction : Bool;
            C17_Slave02_Disconnected : Bool;
            C17_Slave02_Malfunction : Bool;
            C17_Reserved_4 : Bool;
            C17_Reserved_5 : Bool;
            C17_Reserved_6 : Bool;
            C17_Reserved_7 : Bool;
            C17_SenManifold_01_Break : Bool;
            C17_SenManifold_01_Short : Bool;
            C17_SenManifold_02_Break : Bool;
            C17_SenManifold_02_Short : Bool;
            C17_SenManifold_03_Break : Bool;
            C17_SenManifold_03_Short : Bool;
            C17_SenManifold_04_Break : Bool;
            C17_SenManifold_04_Short : Bool;
            C17_IsoVlvSlv_1_Break : Bool;
            C17_IsoVlvSlv_1_Short : Bool;
            C17_IsoVlvSlv_2_Break : Bool;
            C17_IsoVlvSlv_2_Short : Bool;
            C17_DustSensor_1_Break : Bool;
            C17_DustSensor_1_Short : Bool;
            C17_DustSensor_2_Break : Bool;
            C17_DustSensor_2_Short : Bool;
            C17_InDamper_1_NotOpn : Bool;
            C17_InDamper_1_NotCls : Bool;
            C17_InDamper_2_NotOpn : Bool;
            C17_InDamper_2_NotCls : Bool;
            C17_OutDamper_1_NotOpn : Bool;
            C17_OutDamper_1_NotCls : Bool;
            C17_OutDamper_2_NotOpn : Bool;
            C17_OutDamper_2_NotCls : Bool;
            C18_Slave01_Disconnected : Bool;
            C18_Slave01_Malfunction : Bool;
            C18_Slave02_Disconnected : Bool;
            C18_Slave02_Malfunction : Bool;
            C18_Reserved_4 : Bool;
            C18_Reserved_5 : Bool;
            C18_Reserved_6 : Bool;
            C18_Reserved_7 : Bool;
            C18_SenManifold_01_Break : Bool;
            C18_SenManifold_01_Short : Bool;
            C18_SenManifold_02_Break : Bool;
            C18_SenManifold_02_Short : Bool;
            C18_SenManifold_03_Break : Bool;
            C18_SenManifold_03_Short : Bool;
            C18_SenManifold_04_Break : Bool;
            C18_SenManifold_04_Short : Bool;
            C18_IsoVlvSlv_1_Break : Bool;
            C18_IsoVlvSlv_1_Short : Bool;
            C18_IsoVlvSlv_2_Break : Bool;
            C18_IsoVlvSlv_2_Short : Bool;
            C18_DustSensor_1_Break : Bool;
            C18_DustSensor_1_Short : Bool;
            C18_DustSensor_2_Break : Bool;
            C18_DustSensor_2_Short : Bool;
            C18_InDamper_1_NotOpn : Bool;
            C18_InDamper_1_NotCls : Bool;
            C18_InDamper_2_NotOpn : Bool;
            C18_InDamper_2_NotCls : Bool;
            C18_OutDamper_1_NotOpn : Bool;
            C18_OutDamper_1_NotCls : Bool;
            C18_OutDamper_2_NotOpn : Bool;
            C18_OutDamper_2_NotCls : Bool;
            C19_Slave01_Disconnected : Bool;
            C19_Slave01_Malfunction : Bool;
            C19_Slave02_Disconnected : Bool;
            C19_Slave02_Malfunction : Bool;
            C19_Reserved_4 : Bool;
            C19_Reserved_5 : Bool;
            C19_Reserved_6 : Bool;
            C19_Reserved_7 : Bool;
            C19_SenManifold_01_Break : Bool;
            C19_SenManifold_01_Short : Bool;
            C19_SenManifold_02_Break : Bool;
            C19_SenManifold_02_Short : Bool;
            C19_SenManifold_03_Break : Bool;
            C19_SenManifold_03_Short : Bool;
            C19_SenManifold_04_Break : Bool;
            C19_SenManifold_04_Short : Bool;
            C19_IsoVlvSlv_1_Break : Bool;
            C19_IsoVlvSlv_1_Short : Bool;
            C19_IsoVlvSlv_2_Break : Bool;
            C19_IsoVlvSlv_2_Short : Bool;
            C19_DustSensor_1_Break : Bool;
            C19_DustSensor_1_Short : Bool;
            C19_DustSensor_2_Break : Bool;
            C19_DustSensor_2_Short : Bool;
            C19_InDamper_1_NotOpn : Bool;
            C19_InDamper_1_NotCls : Bool;
            C19_InDamper_2_NotOpn : Bool;
            C19_InDamper_2_NotCls : Bool;
            C19_OutDamper_1_NotOpn : Bool;
            C19_OutDamper_1_NotCls : Bool;
            C19_OutDamper_2_NotOpn : Bool;
            C19_OutDamper_2_NotCls : Bool;
            C20_Slave01_Disconnected : Bool;
            C20_Slave01_Malfunction : Bool;
            C20_Slave02_Disconnected : Bool;
            C20_Slave02_Malfunction : Bool;
            C20_Reserved_4 : Bool;
            C20_Reserved_5 : Bool;
            C20_Reserved_6 : Bool;
            C20_Reserved_7 : Bool;
            C20_SenManifold_01_Break : Bool;
            C20_SenManifold_01_Short : Bool;
            C20_SenManifold_02_Break : Bool;
            C20_SenManifold_02_Short : Bool;
            C20_SenManifold_03_Break : Bool;
            C20_SenManifold_03_Short : Bool;
            C20_SenManifold_04_Break : Bool;
            C20_SenManifold_04_Short : Bool;
            C20_IsoVlvSlv_1_Break : Bool;
            C20_IsoVlvSlv_1_Short : Bool;
            C20_IsoVlvSlv_2_Break : Bool;
            C20_IsoVlvSlv_2_Short : Bool;
            C20_DustSensor_1_Break : Bool;
            C20_DustSensor_1_Short : Bool;
            C20_DustSensor_2_Break : Bool;
            C20_DustSensor_2_Short : Bool;
            C20_InDamper_1_NotOpn : Bool;
            C20_InDamper_1_NotCls : Bool;
            C20_InDamper_2_NotOpn : Bool;
            C20_InDamper_2_NotCls : Bool;
            C20_OutDamper_1_NotOpn : Bool;
            C20_OutDamper_1_NotCls : Bool;
            C20_OutDamper_2_NotOpn : Bool;
            C20_OutDamper_2_NotCls : Bool;
            C21_Slave01_Disconnected : Bool;
            C21_Slave01_Malfunction : Bool;
            C21_Slave02_Disconnected : Bool;
            C21_Slave02_Malfunction : Bool;
            C21_Reserved_4 : Bool;
            C21_Reserved_5 : Bool;
            C21_Reserved_6 : Bool;
            C21_Reserved_7 : Bool;
            C21_SenManifold_01_Break : Bool;
            C21_SenManifold_01_Short : Bool;
            C21_SenManifold_02_Break : Bool;
            C21_SenManifold_02_Short : Bool;
            C21_SenManifold_03_Break : Bool;
            C21_SenManifold_03_Short : Bool;
            C21_SenManifold_04_Break : Bool;
            C21_SenManifold_04_Short : Bool;
            C21_IsoVlvSlv_1_Break : Bool;
            C21_IsoVlvSlv_1_Short : Bool;
            C21_IsoVlvSlv_2_Break : Bool;
            C21_IsoVlvSlv_2_Short : Bool;
            C21_DustSensor_1_Break : Bool;
            C21_DustSensor_1_Short : Bool;
            C21_DustSensor_2_Break : Bool;
            C21_DustSensor_2_Short : Bool;
            C21_InDamper_1_NotOpn : Bool;
            C21_InDamper_1_NotCls : Bool;
            C21_InDamper_2_NotOpn : Bool;
            C21_InDamper_2_NotCls : Bool;
            C21_OutDamper_1_NotOpn : Bool;
            C21_OutDamper_1_NotCls : Bool;
            C21_OutDamper_2_NotOpn : Bool;
            C21_OutDamper_2_NotCls : Bool;
            C22_Slave01_Disconnected : Bool;
            C22_Slave01_Malfunction : Bool;
            C22_Slave02_Disconnected : Bool;
            C22_Slave02_Malfunction : Bool;
            C22_Reserved_4 : Bool;
            C22_Reserved_5 : Bool;
            C22_Reserved_6 : Bool;
            C22_Reserved_7 : Bool;
            C22_SenManifold_01_Break : Bool;
            C22_SenManifold_01_Short : Bool;
            C22_SenManifold_02_Break : Bool;
            C22_SenManifold_02_Short : Bool;
            C22_SenManifold_03_Break : Bool;
            C22_SenManifold_03_Short : Bool;
            C22_SenManifold_04_Break : Bool;
            C22_SenManifold_04_Short : Bool;
            C22_IsoVlvSlv_1_Break : Bool;
            C22_IsoVlvSlv_1_Short : Bool;
            C22_IsoVlvSlv_2_Break : Bool;
            C22_IsoVlvSlv_2_Short : Bool;
            C22_DustSensor_1_Break : Bool;
            C22_DustSensor_1_Short : Bool;
            C22_DustSensor_2_Break : Bool;
            C22_DustSensor_2_Short : Bool;
            C22_InDamper_1_NotOpn : Bool;
            C22_InDamper_1_NotCls : Bool;
            C22_InDamper_2_NotOpn : Bool;
            C22_InDamper_2_NotCls : Bool;
            C22_OutDamper_1_NotOpn : Bool;
            C22_OutDamper_1_NotCls : Bool;
            C22_OutDamper_2_NotOpn : Bool;
            C22_OutDamper_2_NotCls : Bool;
            C23_Slave01_Disconnected : Bool;
            C23_Slave01_Malfunction : Bool;
            C23_Slave02_Disconnected : Bool;
            C23_Slave02_Malfunction : Bool;
            C23_Reserved_4 : Bool;
            C23_Reserved_5 : Bool;
            C23_Reserved_6 : Bool;
            C23_Reserved_7 : Bool;
            C23_SenManifold_01_Break : Bool;
            C23_SenManifold_01_Short : Bool;
            C23_SenManifold_02_Break : Bool;
            C23_SenManifold_02_Short : Bool;
            C23_SenManifold_03_Break : Bool;
            C23_SenManifold_03_Short : Bool;
            C23_SenManifold_04_Break : Bool;
            C23_SenManifold_04_Short : Bool;
            C23_IsoVlvSlv_1_Break : Bool;
            C23_IsoVlvSlv_1_Short : Bool;
            C23_IsoVlvSlv_2_Break : Bool;
            C23_IsoVlvSlv_2_Short : Bool;
            C23_DustSensor_1_Break : Bool;
            C23_DustSensor_1_Short : Bool;
            C23_DustSensor_2_Break : Bool;
            C23_DustSensor_2_Short : Bool;
            C23_InDamper_1_NotOpn : Bool;
            C23_InDamper_1_NotCls : Bool;
            C23_InDamper_2_NotOpn : Bool;
            C23_InDamper_2_NotCls : Bool;
            C23_OutDamper_1_NotOpn : Bool;
            C23_OutDamper_1_NotCls : Bool;
            C23_OutDamper_2_NotOpn : Bool;
            C23_OutDamper_2_NotCls : Bool;
            C24_Slave01_Disconnected : Bool;
            C24_Slave01_Malfunction : Bool;
            C24_Slave02_Disconnected : Bool;
            C24_Slave02_Malfunction : Bool;
            C24_Reserved_4 : Bool;
            C24_Reserved_5 : Bool;
            C24_Reserved_6 : Bool;
            C24_Reserved_7 : Bool;
            C24_SenManifold_01_Break : Bool;
            C24_SenManifold_01_Short : Bool;
            C24_SenManifold_02_Break : Bool;
            C24_SenManifold_02_Short : Bool;
            C24_SenManifold_03_Break : Bool;
            C24_SenManifold_03_Short : Bool;
            C24_SenManifold_04_Break : Bool;
            C24_SenManifold_04_Short : Bool;
            C24_IsoVlvSlv_1_Break : Bool;
            C24_IsoVlvSlv_1_Short : Bool;
            C24_IsoVlvSlv_2_Break : Bool;
            C24_IsoVlvSlv_2_Short : Bool;
            C24_DustSensor_1_Break : Bool;
            C24_DustSensor_1_Short : Bool;
            C24_DustSensor_2_Break : Bool;
            C24_DustSensor_2_Short : Bool;
            C24_InDamper_1_NotOpn : Bool;
            C24_InDamper_1_NotCls : Bool;
            C24_InDamper_2_NotOpn : Bool;
            C24_InDamper_2_NotCls : Bool;
            C24_OutDamper_1_NotOpn : Bool;
            C24_OutDamper_1_NotCls : Bool;
            C24_OutDamper_2_NotOpn : Bool;
            C24_OutDamper_2_NotCls : Bool;
         END_STRUCT;
         Header_Info_5 : Byte;
         HE5750_1_AI_Break : Bool;   // User Defined
         HE5750_1_AI_Short : Bool;   // User Defined
         HE5750_2_AI_Break : Bool;   // User Defined
         HE5750_2_AI_Short : Bool;   // User Defined
         HE5750_3_AI_Break : Bool;   // User Defined
         HE5750_3_AI_Short : Bool;   // User Defined
         HE5750_4_AI_Break : Bool;   // User Defined
         HE5750_4_AI_Short : Bool;   // User Defined
         HE5910_1_AI_Break : Bool;   // User Defined
         HE5910_1_AI_Short : Bool;   // User Defined
         HE5910_2_AI_Break : Bool;   // User Defined
         HE5910_2_AI_Short : Bool;   // User Defined
         HE5910_3_AI_Break : Bool;   // User Defined
         HE5910_3_AI_Short : Bool;   // User Defined
         HE5910_4_AI_Break : Bool;   // User Defined
         HE5910_4_AI_Short : Bool;   // User Defined
         FBStorage : Array[0..19] of Byte;
      END_STRUCT;
      TYPE_800_AI_REAL : Array[0..19] of Real;
      ONS : Struct
         AckAlarm : Bool;
         Cmd_Auto : Bool;
         Cmd_Manual : Bool;
         CMD_Local : Bool;
         CMD_Test : Bool;
         GLTP : Bool;
         RET : Bool;
         CMD_Start : Bool;
         FP_Start_CMD : Bool;
         SecPulse1 : Bool;
         SecPulse2 : Bool;
         xTestDamperOpen : Bool;
         xTestDamperClose : Bool;
         xUnlockIsolationValve : Bool;
         xTestInletDamper1 : Bool;
         xTestInletDamper2 : Bool;
         xTestOutletDamper1 : Bool;
         xTestOutletDamper2 : Bool;
         x1691EVOMode : Bool;
         xOfflineCleaning : Bool;
         xSemiOfflineCleaning : Bool;
         xPostCleaning : Bool;
         xForcedCleaning : Bool;
         xDoublePurgeClean : Bool;
      END_STRUCT;
      StatusWork : Int;
      ModePointer : Int;
      AlarmNo : Int;
      AlarmNo_Old : Int;
      StartWarn_Mem : Int;
      RunDelay_Mem : Int;
      DelayStart_Mem : Int;
      DelayStop_Mem : Int;
      ReturnMon_Mem : Int;
      ResetCmd_Mem : Int;
      TimerTestCommand_Mem : Int;
      CompartmentCounter : Byte;
      ModeAuto : Bool;
      ModeLocal : Bool;
      ModeManual : Bool;
      ModeSingleStart : Bool;
      Select : Bool;   // Parent & Program Select
      CMD_AckAlarm : Bool;
      CMD_Start : Bool;
      CMD_Stop : Bool;
      CMD_QStop : Bool;
      CMD_Reset : Bool;
      FromStateAuto : Bool;
      FromStateSingle : Bool;
      FromStateManual : Bool;
      FromStateLocal : Bool;
      FromStopState : Bool;
      ALARM_SupressionActive : Bool;
      ALARM_AlarmPresent : Bool;
      ALARM_WarnPresent : Bool;
      ALARM_FailureAckRequired : Bool;
      ALARM_WarnAckRequired : Bool;
      StartWarn_TT : Bool;
      StartWarn_Done : Bool;
      Rundelay_Done : Bool;
      DelayStart_Done : Bool;
      DelayStop_Done : Bool;
      ReturnMon_Done : Bool;
      Trig_RET_ALARM : Bool;
      RET_OneScan : Bool;
      NotEmpty : Bool;   // Unit Stopped un-normal
      LSTR_Puls : Bool;
      Sec_Pulse : Bool;
      RET : Bool;   // Feedback contact
      GFA : Bool := TRUE;   // General fault
      GWA : Bool := TRUE;   // General waring
      CON : Bool;   // Command 1
      BUSF : Bool := TRUE;   // Bus failure
      Type400 : Bool;   // Filter Type 400
      Type800 : Bool;   // Filter Type 800
      Type_UniClean : Bool;   // Filter Type 1691 - Uni Clean Filter
      Type_FabriClean : Bool;   // Filter Type 1691 - Fabri Clean Filter
      Type1691 : Bool;
      xAlarmReset : Bool;
      ReseTestCommand : Bool;
      DiagBusy : Bool;
      Type820 : Bool;   // Filter type 820
      Type1691EVO : Bool;
      "ONS.xDoublePurgeCleanCCR" : Bool;
      Spare_StatBool : Bool;
      OUT : Struct
         LAMP : Bool;
         SACK : Bool;
         RD : Bool;
         RUN : Bool;
         OK : Bool;
         LOC : Bool;
         MAN : Bool;
         AUT : Bool;
         SS : Bool;
         RES : Bool;
         ASTW : Bool;
         AL_SUPR : Bool;
         FRC_CL : Bool;
         PST_CL : Bool;
         LPA : Bool;
         RLC : Bool;
         SFLT : Bool;
         INTL_OK_STAT : Bool;
         INTL_SEQ_STR_OK_STAT : Bool;
         INTL_SEQ_STP_OK_STAT : Bool;
         "MSW.EXT.AlarmFailUnAck" : Bool;
      END_STRUCT;
      MSW_Status_Trans : Int;
   END_VAR
   VAR_TEMP
      AOn : Bool;   // Always On
      AOff : Bool;   // Always Off
      DummyBool : Bool;
      Temp_CON : Bool;
      ResetCmdDelay_Dn : Bool;
      TempInt : Int;
      StatPointer_Old : Int;
      StatusBuilder : Int;
      bCFG_Chamber : Byte;   // Number of chamber possiblity
      TmpChamberLength : Int;
      TmpIOAddrDigital : Int;
      TmpAnalogLength : Int;
      DiagRetVal : Int;
      wInputIOAddr : Word;   // SPC->PLC Start Address in the Process Image for one SPC WORD FORMAT
      wOutputIOAddr : Word;
      wDigitalIOAddr : Word;
      wChamberLength : Word;
      wAnalogLength : Word;
      wDigitalLength : Word;
      CompartmentOffsetDiag : DWord;
      CompartmentOffset : DWord;
      pSPC_PTRInput : ANY;   // Pointer for SPC Generic Input IO Area
      pSPC_PTROutput : ANY;   // Pointer for SPC Generic Output IO Area
      pSPC_PTRAnalog : ANY;
      pSPC_PTRDigital : ANY;
      pSPC_PTRChambers : ANY;
      pSPC_Device_CompView : ANY;
      pSPC_DiagnosticSystem : ANY;
      pSPC_DiagnosticComp : ANY;
      pSPC_DiagnosticAnalog : ANY;
      MemoryPool_cmd_FINAL : Struct   // This memory will be copied to the OB1 image
         xFilterStart : Bool;
         xFilterStop : Bool;
         xEmergencyStop : Bool;
         xAlarmReset : Bool;
         xOfflineCleaning : Bool;
         xPostCleaning : Bool;
         xForcedCleaning : Bool;
         xSemiOfflineCleaning : Bool;
         LocalControlDisable : Bool;
         RemoteControl : Bool;
         OverwriteComp : Bool;
         x1691EV0Mode : Bool;
         xDoublePurgeClean : Bool;
         xDoublePurgeCleanCCR : Bool;
         xCommandDummy1_6 : Bool;
         xCommandDummy1_7 : Bool;
         xCloseC1 : Bool;
         xCloseC2 : Bool;
         xCloseC3 : Bool;
         xCloseC4 : Bool;
         xCloseC5 : Bool;
         xCloseC6 : Bool;
         xCloseC7 : Bool;
         xCloseC8 : Bool;
         xCloseC9 : Bool;
         xCloseC10 : Bool;
         xCloseC11 : Bool;
         xCloseC12 : Bool;
         xCloseC13 : Bool;
         xCloseC14 : Bool;
         xCloseC15 : Bool;
         xCloseC16 : Bool;
         xCloseC17 : Bool;
         xCloseC18 : Bool;
         xCloseC19 : Bool;
         xCloseC20 : Bool;
         xCloseC21 : Bool;
         xCloseC22 : Bool;
         xCloseC23 : Bool;
         xCloseC24 : Bool;
         xCleanC1 : Bool;
         xCleanC2 : Bool;
         xCleanC3 : Bool;
         xCleanC4 : Bool;
         xCleanC5 : Bool;
         xCleanC6 : Bool;
         xCleanC7 : Bool;
         xCleanC8 : Bool;
         xCleanC9 : Bool;
         xCleanC10 : Bool;
         xCleanC11 : Bool;
         xCleanC12 : Bool;
         xCleanC13 : Bool;
         xCleanC14 : Bool;
         xCleanC15 : Bool;
         xCleanC16 : Bool;
         xCleanC17 : Bool;
         xCleanC18 : Bool;
         xCleanC19 : Bool;
         xCleanC20 : Bool;
         xCleanC21 : Bool;
         xCleanC22 : Bool;
         xCleanC23 : Bool;
         xCleanC24 : Bool;
         xDELTAP_lower_Offset : Int;
         xDELTAP_higher_Offset : Int;
         xEXTRA_Pause1 : Int;
         xEXTRA_Pause2 : Int;
         xReserved16 : Byte;
         xReserved17 : Byte;
         xReserved18 : Byte;
         xReserved19 : Byte;
         xTestCommandValue : Byte;
         xTestCompartmentNo : Byte;
         xTestValveNo : Byte;
         xTestInletDamper1 : Bool;
         xTestInletDamper2 : Bool;
         xTestOutletDamper1 : Bool;
         xTestOutletDamper2 : Bool;
         xTestDamperDirection : Bool;
         xUnlockIsolationValve : Bool;
         xReserved24 : Byte;
         xReserved25 : Byte;
         xReserved26 : Byte;
         xReserved27 : Byte;
         xReserved28 : Byte;
         xReserved29 : Byte;
         VolumeFlow : Int;
         xReserved32 : Int;
         xReserved34 : Int;
         xReserved36 : Int;
      END_STRUCT;
      CompartmentErrorPointer : Byte;
      pSPC_CompartmentError : ANY;
      BlkRet1 : Int;   // Temporary Return Value
      BlkRet2 : Int;
      BlkRet3 : Int;
      BlkRet4 : Int;
      BlkRet5 : Int;
      BlkRet6 : Int;
      BlkRet7 : Int;
      BlkRet8 : Int;
      BlkRet9 : Int;
      HeaderOffset : Byte;
      NO_AI_Internal : Int;   // Enter number of analog option card normally HE5910
      NO_DI_Internal : Int;   // Enter number of digital option card normally HE5910
      TempDword : DWord;
      TempReal : Real;
      HW_ID : Hw_Any;
      GEOADDR_HW : GEOADDR;
      Status_Add : Int;
   END_VAR
   VAR_TEMP   // added for the SCL form of the ladder/FBD networks
      _w1 : Bool;
      _w2 : Bool;
      _w3 : Bool;
      _w4 : Bool;
      _w5 : Bool;
      _w6 : Bool;
   END_VAR
BEGIN

REGION Network 1: Always On
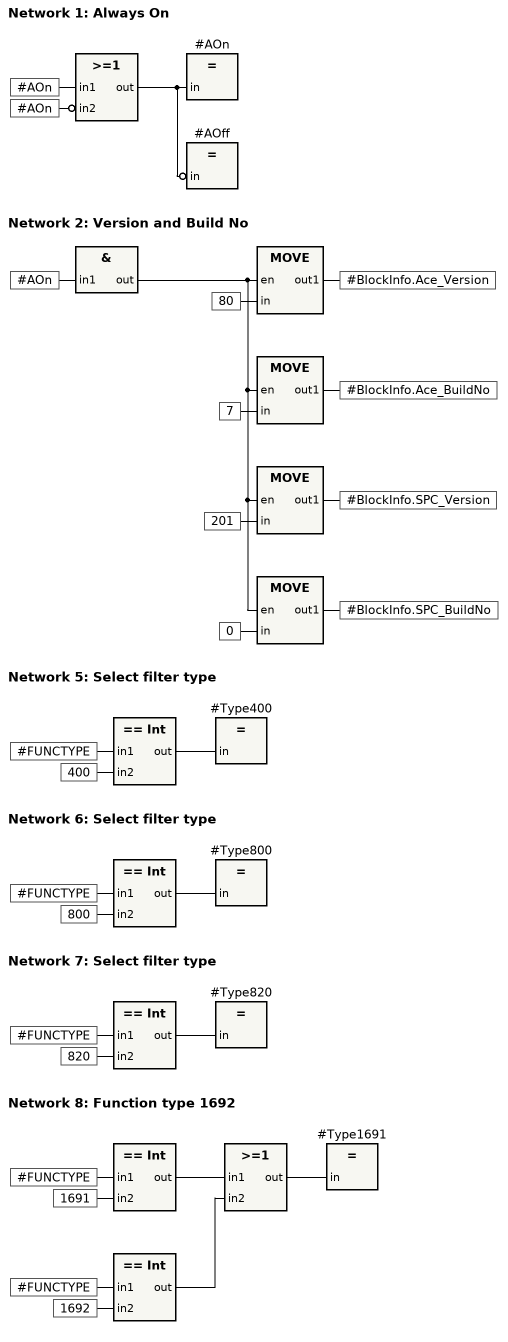
   #AOn := #AOn OR NOT #AOn;
   #AOff := NOT #AOn;
END_REGION

REGION Network 2: Version and Build No
   IF #AOn THEN
       #BlockInfo.Ace_Version := 80;
       #BlockInfo.Ace_BuildNo := 7;
       #BlockInfo.SPC_Version := 201;
       #BlockInfo.SPC_BuildNo := 0;
   END_IF;
END_REGION

REGION Network 3 (STL): Instance DB Number to Faceplate
         L     DINO;
         T     #BlockInfo.DB_Number;
END_REGION

REGION Network 4 (SCL): Transfer Interlock OK to Stat
   #OUT.INTL_OK_STAT := PEEK_BOOL(area := 16#84, dbNumber := #BlockInfo.DB_Number, byteOffset := 24, bitOffset := 0);
   #OUT.INTL_SEQ_STR_OK_STAT := PEEK_BOOL(area := 16#84, dbNumber := #BlockInfo.DB_Number, byteOffset := 26, bitOffset := 0);
   #OUT.INTL_SEQ_STP_OK_STAT := PEEK_BOOL(area := 16#84, dbNumber := #BlockInfo.DB_Number, byteOffset := 28, bitOffset := 0);
END_REGION

REGION Network 5: Select filter type
   #Type400 := #FUNCTYPE = 400;
END_REGION

REGION Network 6: Select filter type
   #Type800 := #FUNCTYPE = 800;
END_REGION

REGION Network 7: Select filter type
   #Type820 := #FUNCTYPE = 820;
END_REGION

REGION Network 8: Function type 1692
   // Build 007 03.12.2020 (VIV-IN) Function Type 1692 added
   #Type1691 := (#FUNCTYPE = 1691) OR (#FUNCTYPE = 1692);
END_REGION

REGION Network 9: Type 1691 EVO
   // Build 007 03.12.2020 (VIV-IN) Type 1691 EVO  Added
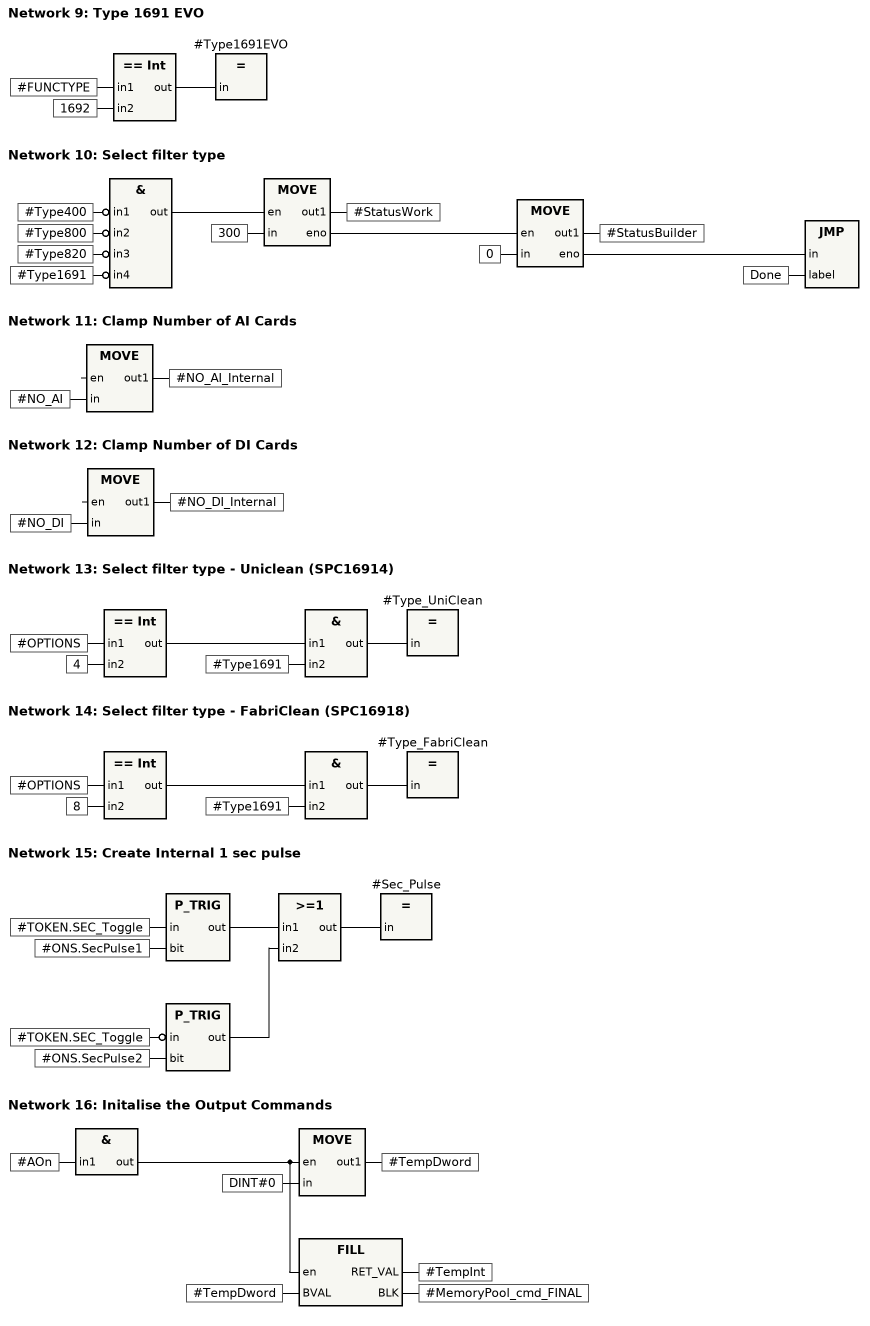
   #Type1691EVO := #FUNCTYPE = 1692;
END_REGION

REGION Network 10: Select filter type
   // ENO of a box is taken as its EN; it also drops when the box reports an error
   #_w1 := NOT #Type400 AND NOT #Type800 AND NOT #Type820 AND NOT #Type1691;
   IF #_w1 THEN
       #StatusWork := 300;
       #StatusBuilder := 0;
       GOTO Done;
   END_IF;
END_REGION

REGION Network 11: Clamp Number of AI Cards
   #NO_AI_Internal := #NO_AI;
END_REGION

REGION Network 12: Clamp Number of DI Cards
   #NO_DI_Internal := #NO_DI;
END_REGION

REGION Network 13: Select filter type - Uniclean (SPC16914)
   // - FilterType for 400/16914 = 400
   #Type_UniClean := (#OPTIONS = 4) AND #Type1691;
END_REGION

REGION Network 14: Select filter type - FabriClean (SPC16918)
   // - FilterType for 800/16918 = 800
   #Type_FabriClean := (#OPTIONS = 8) AND #Type1691;
END_REGION

REGION Network 15: Create Internal 1 sec pulse
   #_w1 := #TOKEN.SEC_Toggle AND NOT #ONS.SecPulse1;   // rising edge
   #ONS.SecPulse1 := #TOKEN.SEC_Toggle;
   #_w2 := NOT #TOKEN.SEC_Toggle AND NOT #ONS.SecPulse2;   // rising edge
   #ONS.SecPulse2 := NOT #TOKEN.SEC_Toggle;
   #Sec_Pulse := #_w1 OR #_w2;
END_REGION

REGION Network 16: Initalise the Output Commands
   IF #AOn THEN
       #TempDword := DINT#0;
       #TempInt := FILL(BVAL := #TempDword, BLK => #MemoryPool_cmd_FINAL);
   END_IF;
END_REGION

REGION Network 17: SET SHOW PARAMETERS
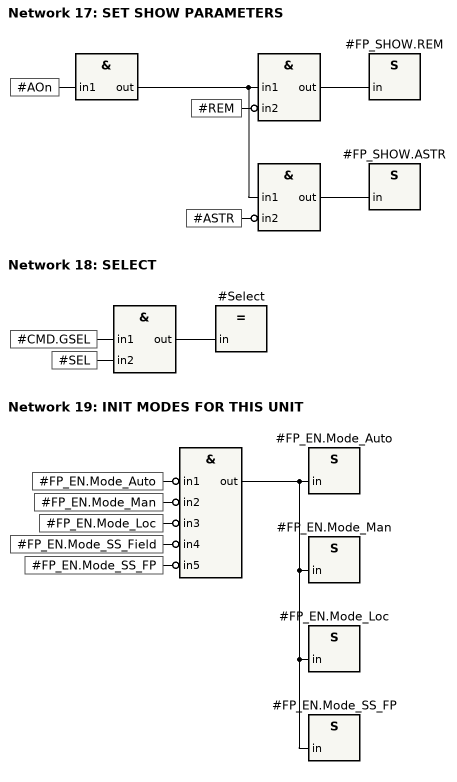
   IF #AOn AND NOT #REM THEN #FP_SHOW.REM := TRUE; END_IF;
   IF #AOn AND NOT #ASTR THEN #FP_SHOW.ASTR := TRUE; END_IF;
END_REGION

REGION Network 18: SELECT
   #Select := #CMD.GSEL AND #SEL;
END_REGION

REGION Network 19: INIT MODES FOR THIS UNIT
   #_w1 := NOT #FP_EN.Mode_Auto AND NOT #FP_EN.Mode_Man AND NOT #FP_EN.Mode_Loc AND NOT #FP_EN.Mode_SS_Field AND NOT #FP_EN.Mode_SS_FP;
   IF #_w1 THEN
       #FP_EN.Mode_Auto := TRUE;
       #FP_EN.Mode_Man := TRUE;
       #FP_EN.Mode_Loc := TRUE;
       #FP_EN.Mode_SS_FP := TRUE;
   END_IF;
END_REGION

REGION Network 20: SHOW PUSH BUTTONS ON FACEPLATE
   // Build 002 - 27 March 2019 : Loc_type flag removed from Show_local
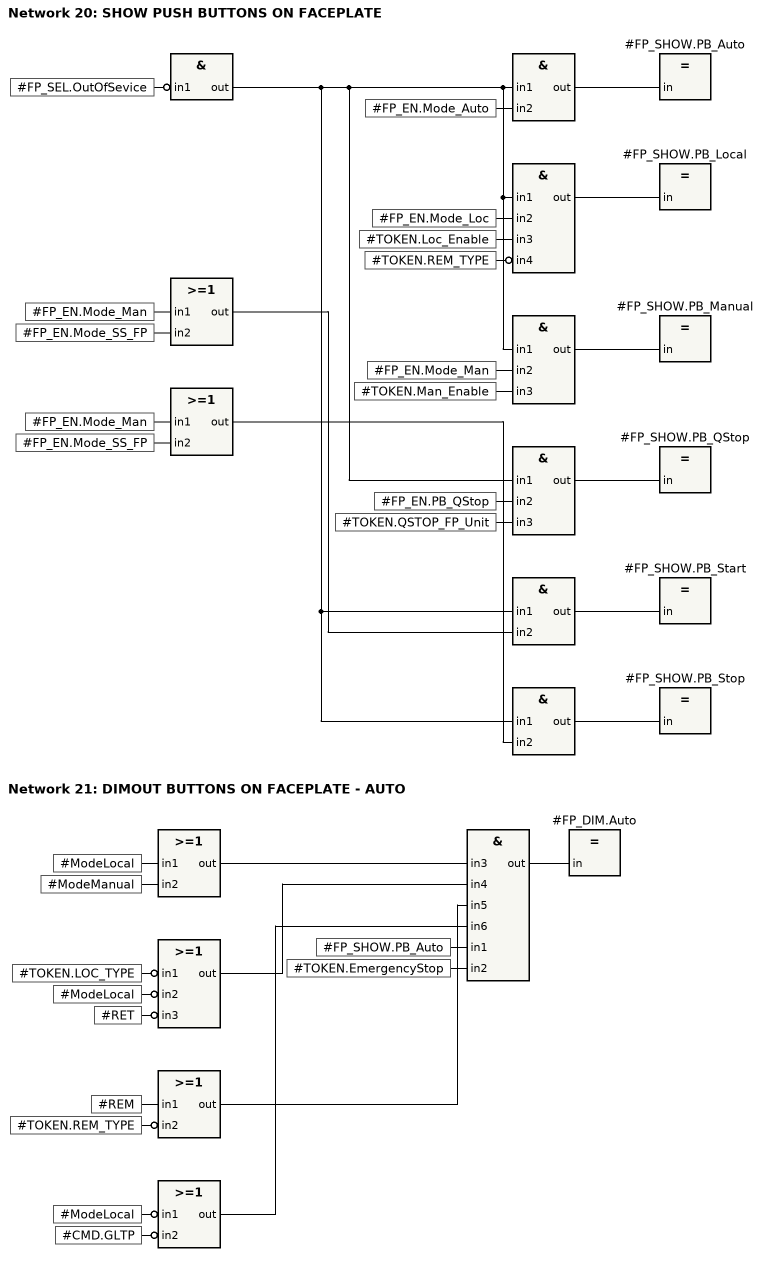
   #FP_SHOW.PB_Auto := NOT #FP_SEL.OutOfSevice AND #FP_EN.Mode_Auto;
   #FP_SHOW.PB_Local := NOT #FP_SEL.OutOfSevice AND #FP_EN.Mode_Loc AND #TOKEN.Loc_Enable AND NOT #TOKEN.REM_TYPE;
   #FP_SHOW.PB_Manual := NOT #FP_SEL.OutOfSevice AND #FP_EN.Mode_Man AND #TOKEN.Man_Enable;
   #FP_SHOW.PB_QStop := NOT #FP_SEL.OutOfSevice AND #FP_EN.PB_QStop AND #TOKEN.QSTOP_FP_Unit;
   #FP_SHOW.PB_Start := NOT #FP_SEL.OutOfSevice AND (#FP_EN.Mode_Man OR #FP_EN.Mode_SS_FP);
   #FP_SHOW.PB_Stop := NOT #FP_SEL.OutOfSevice AND (#FP_EN.Mode_Man OR #FP_EN.Mode_SS_FP);
END_REGION

REGION Network 21: DIMOUT BUTTONS ON FACEPLATE - AUTO
   #FP_DIM.Auto := (#ModeLocal OR #ModeManual) AND (NOT #TOKEN.LOC_TYPE OR NOT #ModeLocal OR NOT #RET) AND (#REM OR NOT #TOKEN.REM_TYPE) AND (NOT #ModeLocal OR NOT #CMD.GLTP) AND #FP_SHOW.PB_Auto AND #TOKEN.EmergencyStop;
END_REGION

REGION Network 22: DIMOUT BUTTONS ON FACEPLATE - MANUAL
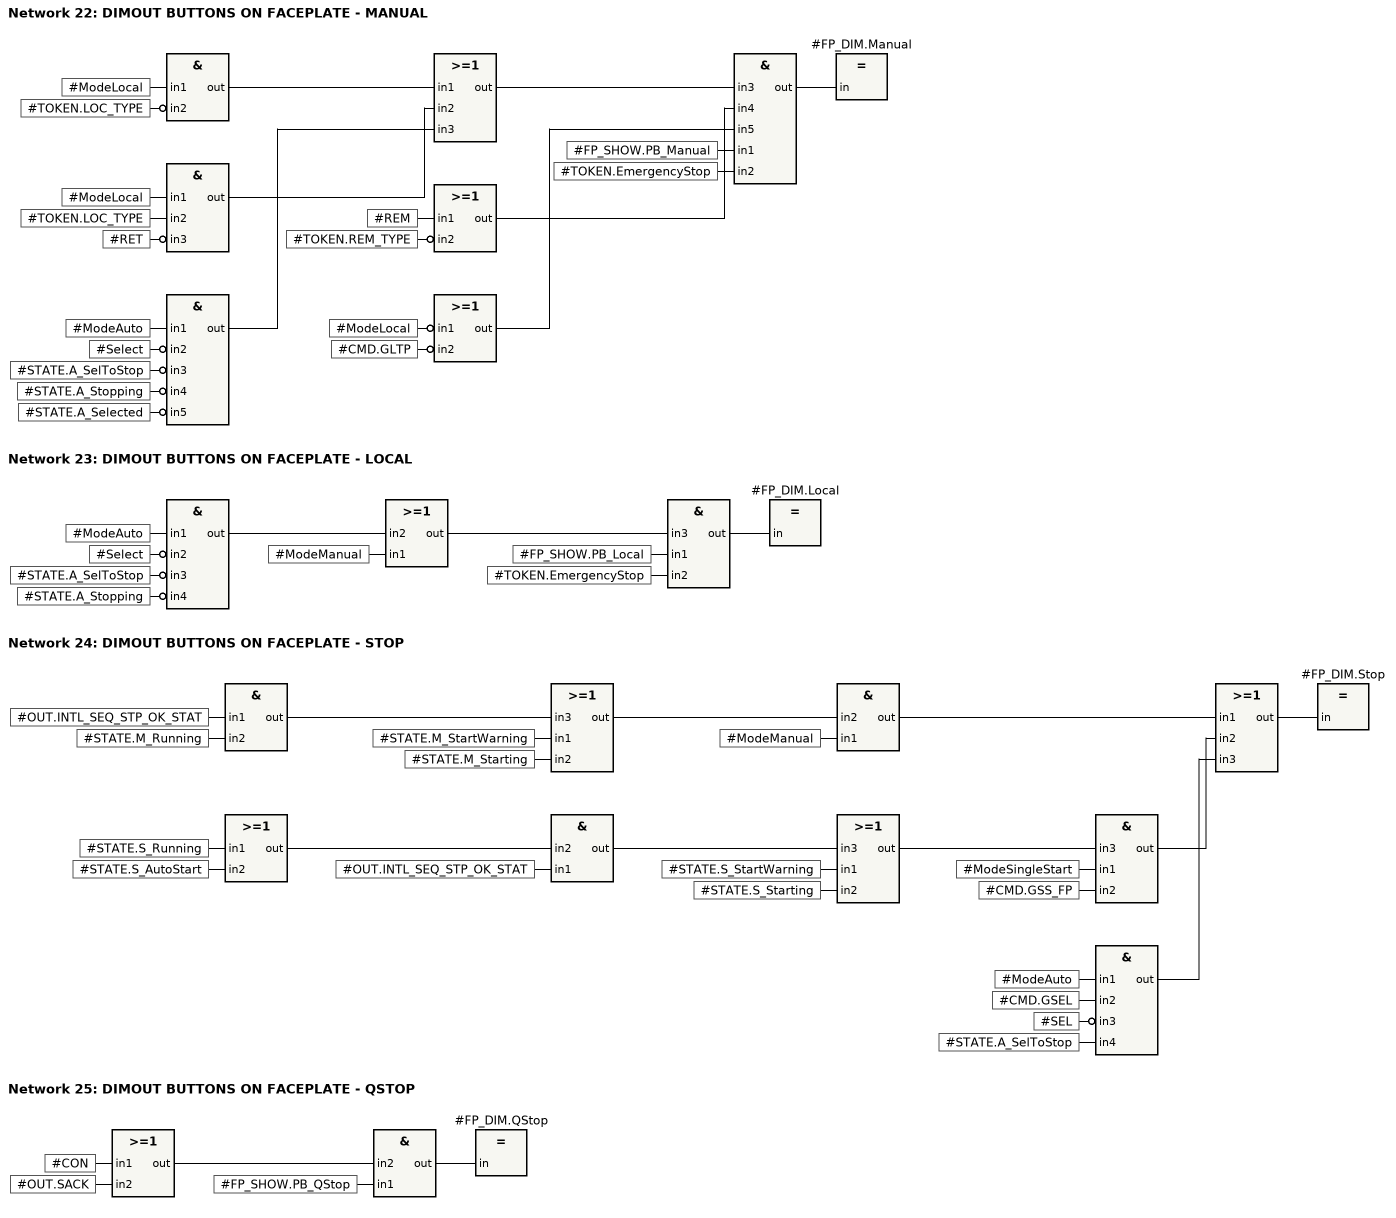
   #FP_DIM.Manual := ((#ModeLocal AND NOT #TOKEN.LOC_TYPE) OR (#ModeLocal AND #TOKEN.LOC_TYPE AND NOT #RET) OR (#ModeAuto AND NOT #Select AND NOT #STATE.A_SelToStop AND NOT #STATE.A_Stopping AND NOT #STATE.A_Selected)) AND (#REM OR NOT #TOKEN.REM_TYPE) AND (NOT #ModeLocal OR NOT #CMD.GLTP) AND #FP_SHOW.PB_Manual AND #TOKEN.EmergencyStop;
END_REGION

REGION Network 23: DIMOUT BUTTONS ON FACEPLATE - LOCAL
   #FP_DIM.Local := ((#ModeAuto AND NOT #Select AND NOT #STATE.A_SelToStop AND NOT #STATE.A_Stopping) OR #ModeManual) AND #FP_SHOW.PB_Local AND #TOKEN.EmergencyStop;
END_REGION

REGION Network 24: DIMOUT BUTTONS ON FACEPLATE - STOP
   #FP_DIM.Stop := (((#OUT.INTL_SEQ_STP_OK_STAT AND #STATE.M_Running) OR #STATE.M_StartWarning OR #STATE.M_Starting) AND #ModeManual) OR ((((#STATE.S_Running OR #STATE.S_AutoStart) AND #OUT.INTL_SEQ_STP_OK_STAT) OR #STATE.S_StartWarning OR #STATE.S_Starting) AND #ModeSingleStart AND #CMD.GSS_FP) OR (#ModeAuto AND #CMD.GSEL AND NOT #SEL AND #STATE.A_SelToStop);
END_REGION

REGION Network 25: DIMOUT BUTTONS ON FACEPLATE - QSTOP
   #FP_DIM.QStop := (#CON OR #OUT.SACK) AND #FP_SHOW.PB_QStop;
END_REGION

REGION Network 26: DIMOUT BUTTONS ON FACEPLATE - START
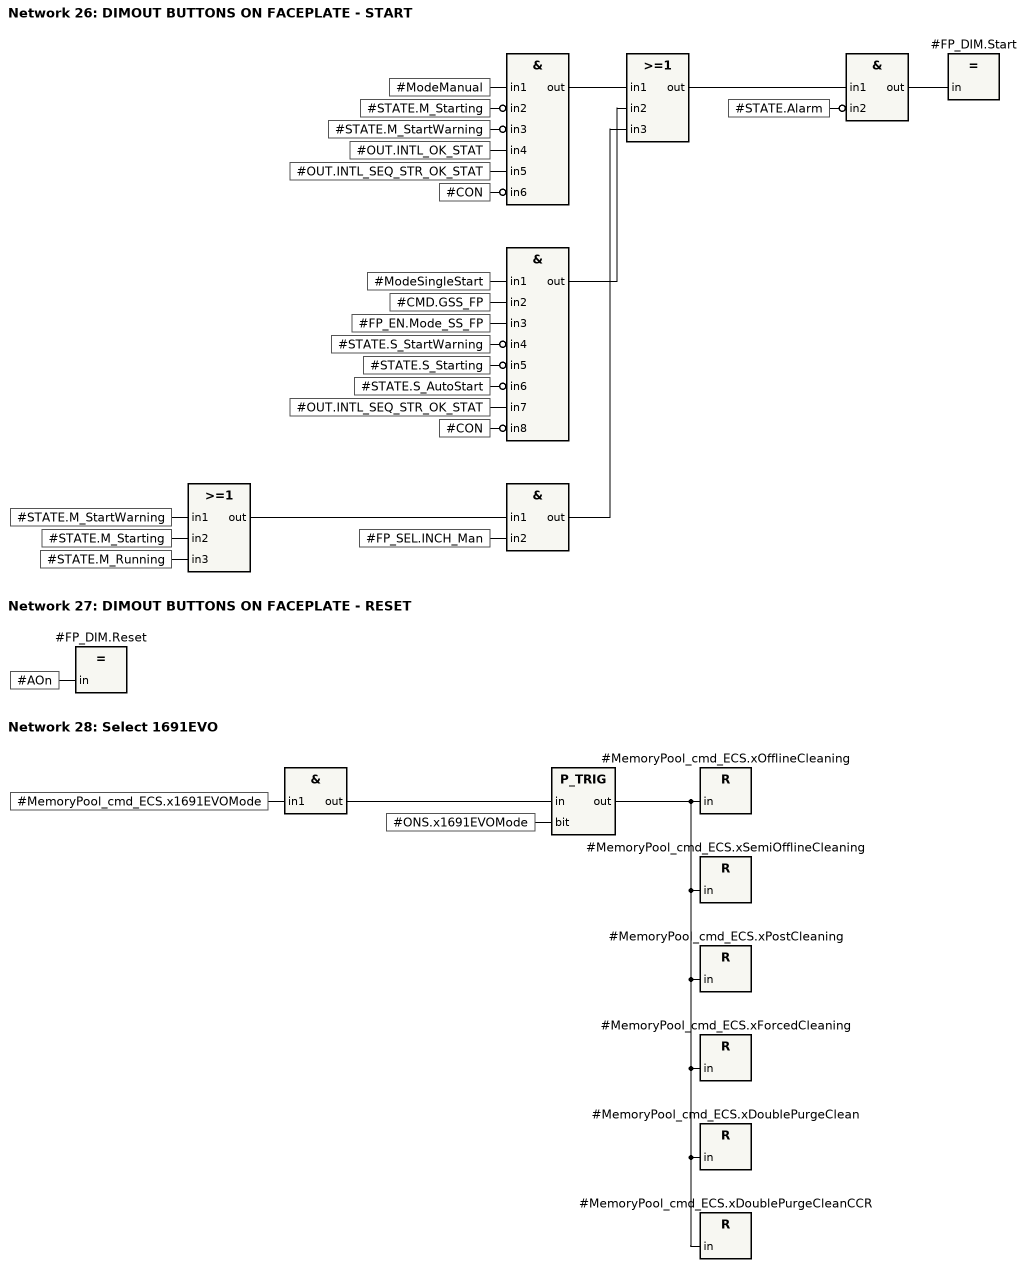
   #FP_DIM.Start := ((#ModeManual AND NOT #STATE.M_Starting AND NOT #STATE.M_StartWarning AND #OUT.INTL_OK_STAT AND #OUT.INTL_SEQ_STR_OK_STAT AND NOT #CON) OR (#ModeSingleStart AND #CMD.GSS_FP AND #FP_EN.Mode_SS_FP AND NOT #STATE.S_StartWarning AND NOT #STATE.S_Starting AND NOT #STATE.S_AutoStart AND #OUT.INTL_SEQ_STR_OK_STAT AND NOT #CON) OR ((#STATE.M_StartWarning OR #STATE.M_Starting OR #STATE.M_Running) AND #FP_SEL.INCH_Man)) AND NOT #STATE.Alarm;
END_REGION

REGION Network 27: DIMOUT BUTTONS ON FACEPLATE - RESET
   #FP_DIM.Reset := #AOn;
END_REGION

REGION Network 28: Select 1691EVO
   // Build 007 - 03.12.2020 (VIV-IN): SPC EVO Type added for FuncType = 1692 
   // Newly Added to deselect other modes if EVO mode Selected
   #_w1 := #MemoryPool_cmd_ECS.x1691EVOMode AND NOT #ONS.x1691EVOMode;   // rising edge
   #ONS.x1691EVOMode := #MemoryPool_cmd_ECS.x1691EVOMode;
   IF #_w1 THEN
       #MemoryPool_cmd_ECS.xOfflineCleaning := FALSE;
       #MemoryPool_cmd_ECS.xSemiOfflineCleaning := FALSE;
       #MemoryPool_cmd_ECS.xPostCleaning := FALSE;
       #MemoryPool_cmd_ECS.xForcedCleaning := FALSE;
       #MemoryPool_cmd_ECS.xDoublePurgeClean := FALSE;
       #MemoryPool_cmd_ECS.xDoublePurgeCleanCCR := FALSE;
   END_IF;
END_REGION

REGION Network 29: Select Double Purge Cleaning
   // Build 007 - 03.12.2020 (VIV-IN): SPC EVO Type added for FuncType = 1692 
   // Newly Added to deselect other modes if Double Purge Selected
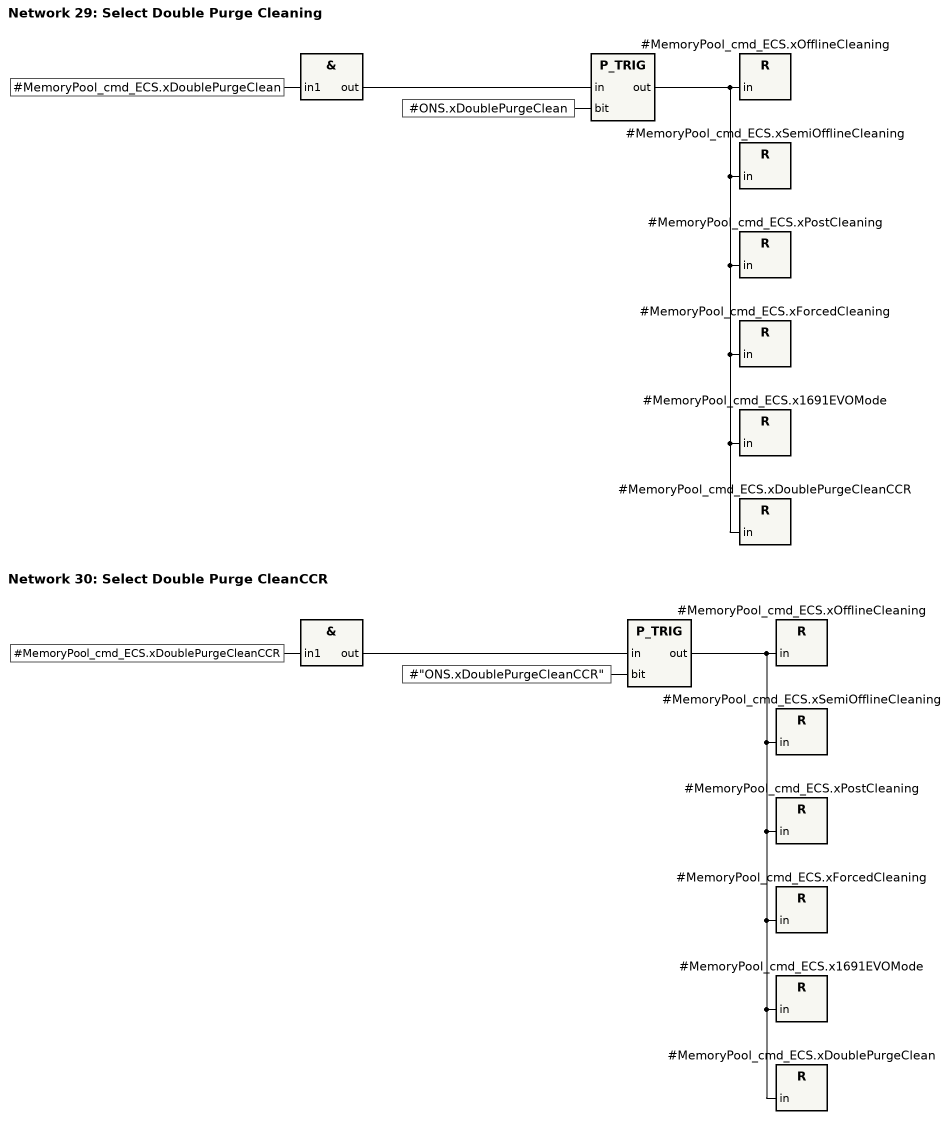
   #_w1 := #MemoryPool_cmd_ECS.xDoublePurgeClean AND NOT #ONS.xDoublePurgeClean;   // rising edge
   #ONS.xDoublePurgeClean := #MemoryPool_cmd_ECS.xDoublePurgeClean;
   IF #_w1 THEN
       #MemoryPool_cmd_ECS.xOfflineCleaning := FALSE;
       #MemoryPool_cmd_ECS.xSemiOfflineCleaning := FALSE;
       #MemoryPool_cmd_ECS.xPostCleaning := FALSE;
       #MemoryPool_cmd_ECS.xForcedCleaning := FALSE;
       #MemoryPool_cmd_ECS.x1691EVOMode := FALSE;
       #MemoryPool_cmd_ECS.xDoublePurgeCleanCCR := FALSE;
   END_IF;
END_REGION

REGION Network 30: Select Double Purge CleanCCR
   // Build 007 - 03.12.2020 (VIV-IN): SPC EVO Type added for FuncType = 1692 
   // Newly Added to deselect other modes if Double Purge CCR Selected
   #_w1 := #MemoryPool_cmd_ECS.xDoublePurgeCleanCCR AND NOT #"ONS.xDoublePurgeCleanCCR";   // rising edge
   #"ONS.xDoublePurgeCleanCCR" := #MemoryPool_cmd_ECS.xDoublePurgeCleanCCR;
   IF #_w1 THEN
       #MemoryPool_cmd_ECS.xOfflineCleaning := FALSE;
       #MemoryPool_cmd_ECS.xSemiOfflineCleaning := FALSE;
       #MemoryPool_cmd_ECS.xPostCleaning := FALSE;
       #MemoryPool_cmd_ECS.xForcedCleaning := FALSE;
       #MemoryPool_cmd_ECS.x1691EVOMode := FALSE;
       #MemoryPool_cmd_ECS.xDoublePurgeClean := FALSE;
   END_IF;
END_REGION

REGION Network 31: Select Offline Cleaning
   // Build 007 - 03.12.2020 (VIV-IN): SPC EVO Type added for FuncType = 1692 
   // Newly Added to deselect other modes if Offline Cleaning Selected
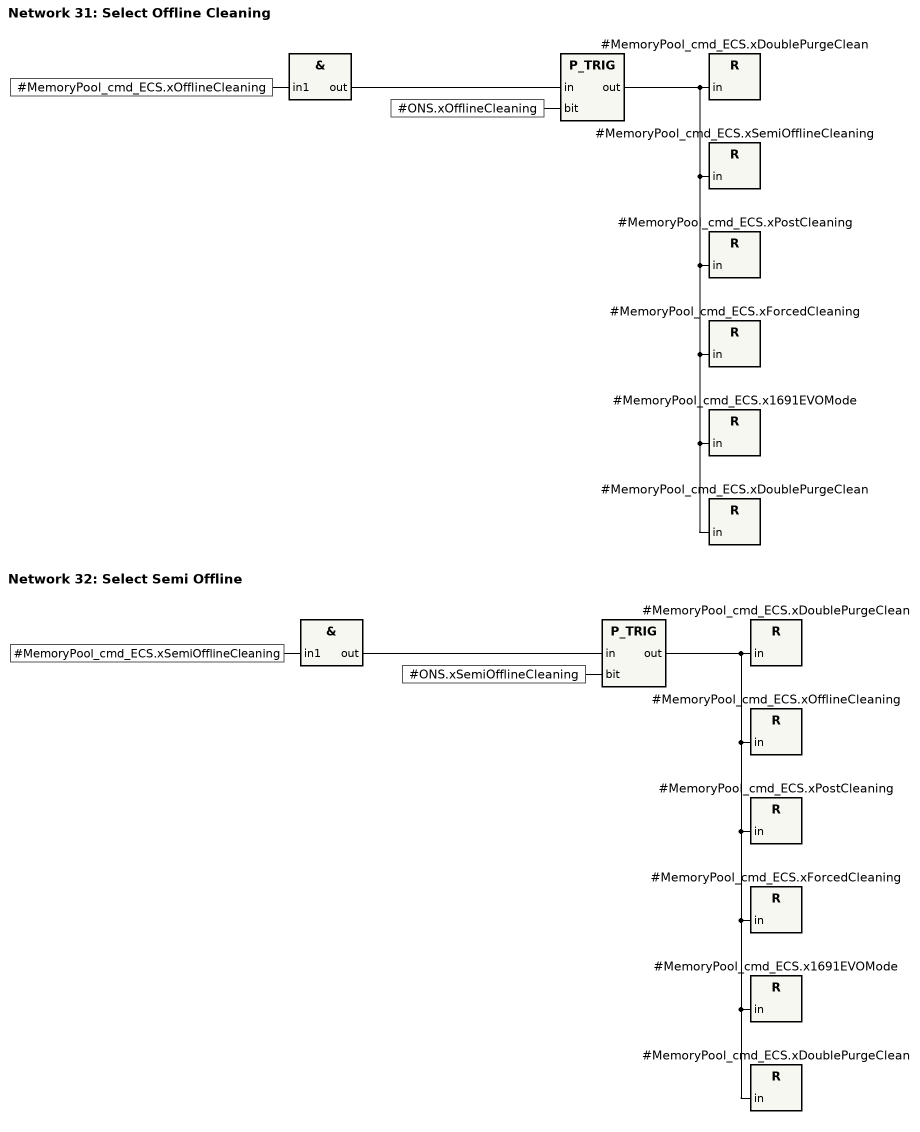
   #_w1 := #MemoryPool_cmd_ECS.xOfflineCleaning AND NOT #ONS.xOfflineCleaning;   // rising edge
   #ONS.xOfflineCleaning := #MemoryPool_cmd_ECS.xOfflineCleaning;
   IF #_w1 THEN
       #MemoryPool_cmd_ECS.xDoublePurgeClean := FALSE;
       #MemoryPool_cmd_ECS.xSemiOfflineCleaning := FALSE;
       #MemoryPool_cmd_ECS.xPostCleaning := FALSE;
       #MemoryPool_cmd_ECS.xForcedCleaning := FALSE;
       #MemoryPool_cmd_ECS.x1691EVOMode := FALSE;
       #MemoryPool_cmd_ECS.xDoublePurgeClean := FALSE;
   END_IF;
END_REGION

REGION Network 32: Select Semi Offline
   // Build 007 - 03.12.2020 (VIV-IN): SPC EVO Type added for FuncType = 1692 
   // Newly Added to deselect other modes if Semi Offline Cleaning Selected
   #_w1 := #MemoryPool_cmd_ECS.xSemiOfflineCleaning AND NOT #ONS.xSemiOfflineCleaning;   // rising edge
   #ONS.xSemiOfflineCleaning := #MemoryPool_cmd_ECS.xSemiOfflineCleaning;
   IF #_w1 THEN
       #MemoryPool_cmd_ECS.xDoublePurgeClean := FALSE;
       #MemoryPool_cmd_ECS.xOfflineCleaning := FALSE;
       #MemoryPool_cmd_ECS.xPostCleaning := FALSE;
       #MemoryPool_cmd_ECS.xForcedCleaning := FALSE;
       #MemoryPool_cmd_ECS.x1691EVOMode := FALSE;
       #MemoryPool_cmd_ECS.xDoublePurgeClean := FALSE;
   END_IF;
END_REGION

REGION Network 33: Select Post cleaning
   // Build 007 - 03.12.2020 (VIV-IN): SPC EVO Type added for FuncType = 1692 
   // Newly Added to deselect other modes if Post Cleaning Selected
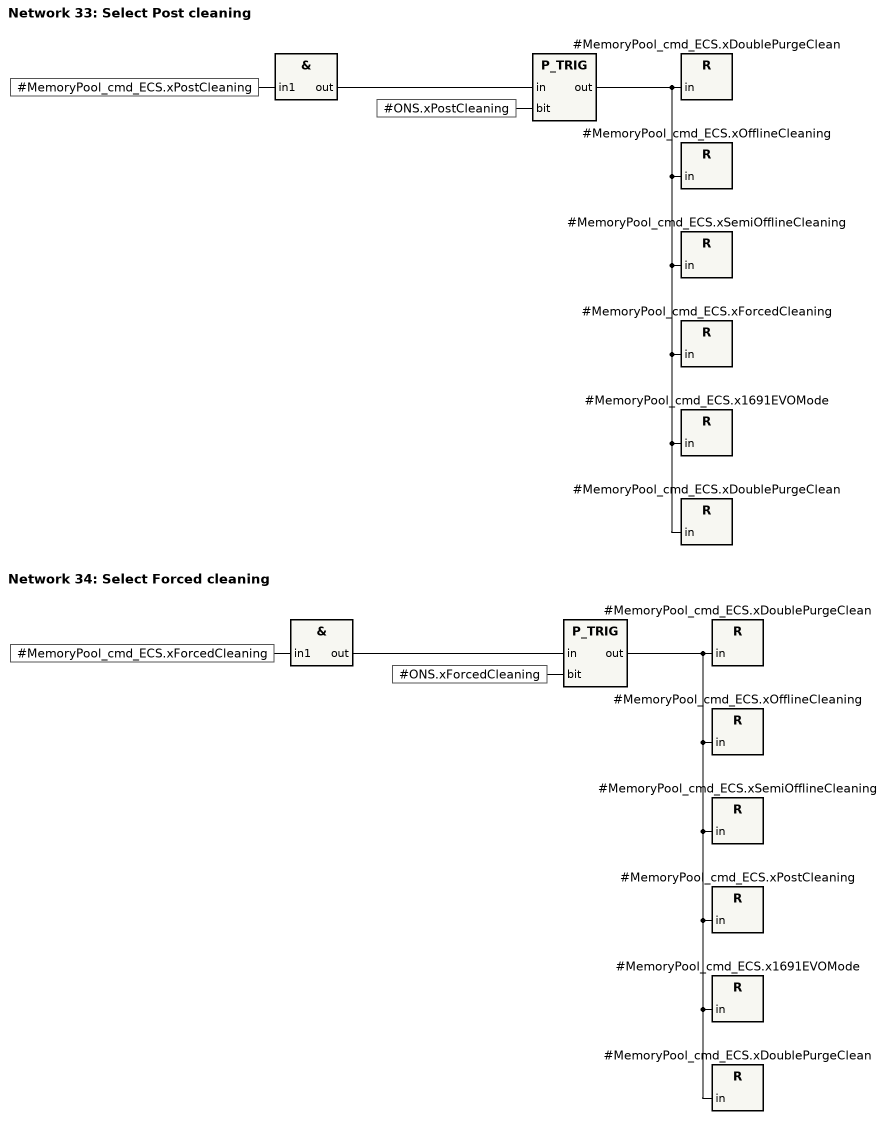
   #_w1 := #MemoryPool_cmd_ECS.xPostCleaning AND NOT #ONS.xPostCleaning;   // rising edge
   #ONS.xPostCleaning := #MemoryPool_cmd_ECS.xPostCleaning;
   IF #_w1 THEN
       #MemoryPool_cmd_ECS.xDoublePurgeClean := FALSE;
       #MemoryPool_cmd_ECS.xOfflineCleaning := FALSE;
       #MemoryPool_cmd_ECS.xSemiOfflineCleaning := FALSE;
       #MemoryPool_cmd_ECS.xForcedCleaning := FALSE;
       #MemoryPool_cmd_ECS.x1691EVOMode := FALSE;
       #MemoryPool_cmd_ECS.xDoublePurgeClean := FALSE;
   END_IF;
END_REGION

REGION Network 34: Select Forced cleaning
   // Build 007 - 03.12.2020 (VIV-IN): SPC EVO Type added for FuncType = 1692 
   // Newly Added to deselect other modes if Forced Cleaning Selected
   #_w1 := #MemoryPool_cmd_ECS.xForcedCleaning AND NOT #ONS.xForcedCleaning;   // rising edge
   #ONS.xForcedCleaning := #MemoryPool_cmd_ECS.xForcedCleaning;
   IF #_w1 THEN
       #MemoryPool_cmd_ECS.xDoublePurgeClean := FALSE;
       #MemoryPool_cmd_ECS.xOfflineCleaning := FALSE;
       #MemoryPool_cmd_ECS.xSemiOfflineCleaning := FALSE;
       #MemoryPool_cmd_ECS.xPostCleaning := FALSE;
       #MemoryPool_cmd_ECS.x1691EVOMode := FALSE;
       #MemoryPool_cmd_ECS.xDoublePurgeClean := FALSE;
   END_IF;
END_REGION

REGION Network 35: MODE Handling - Auto Mode
   // Build 002 - 27 March 2019: REM flag is removed in FP_CMD.Auto
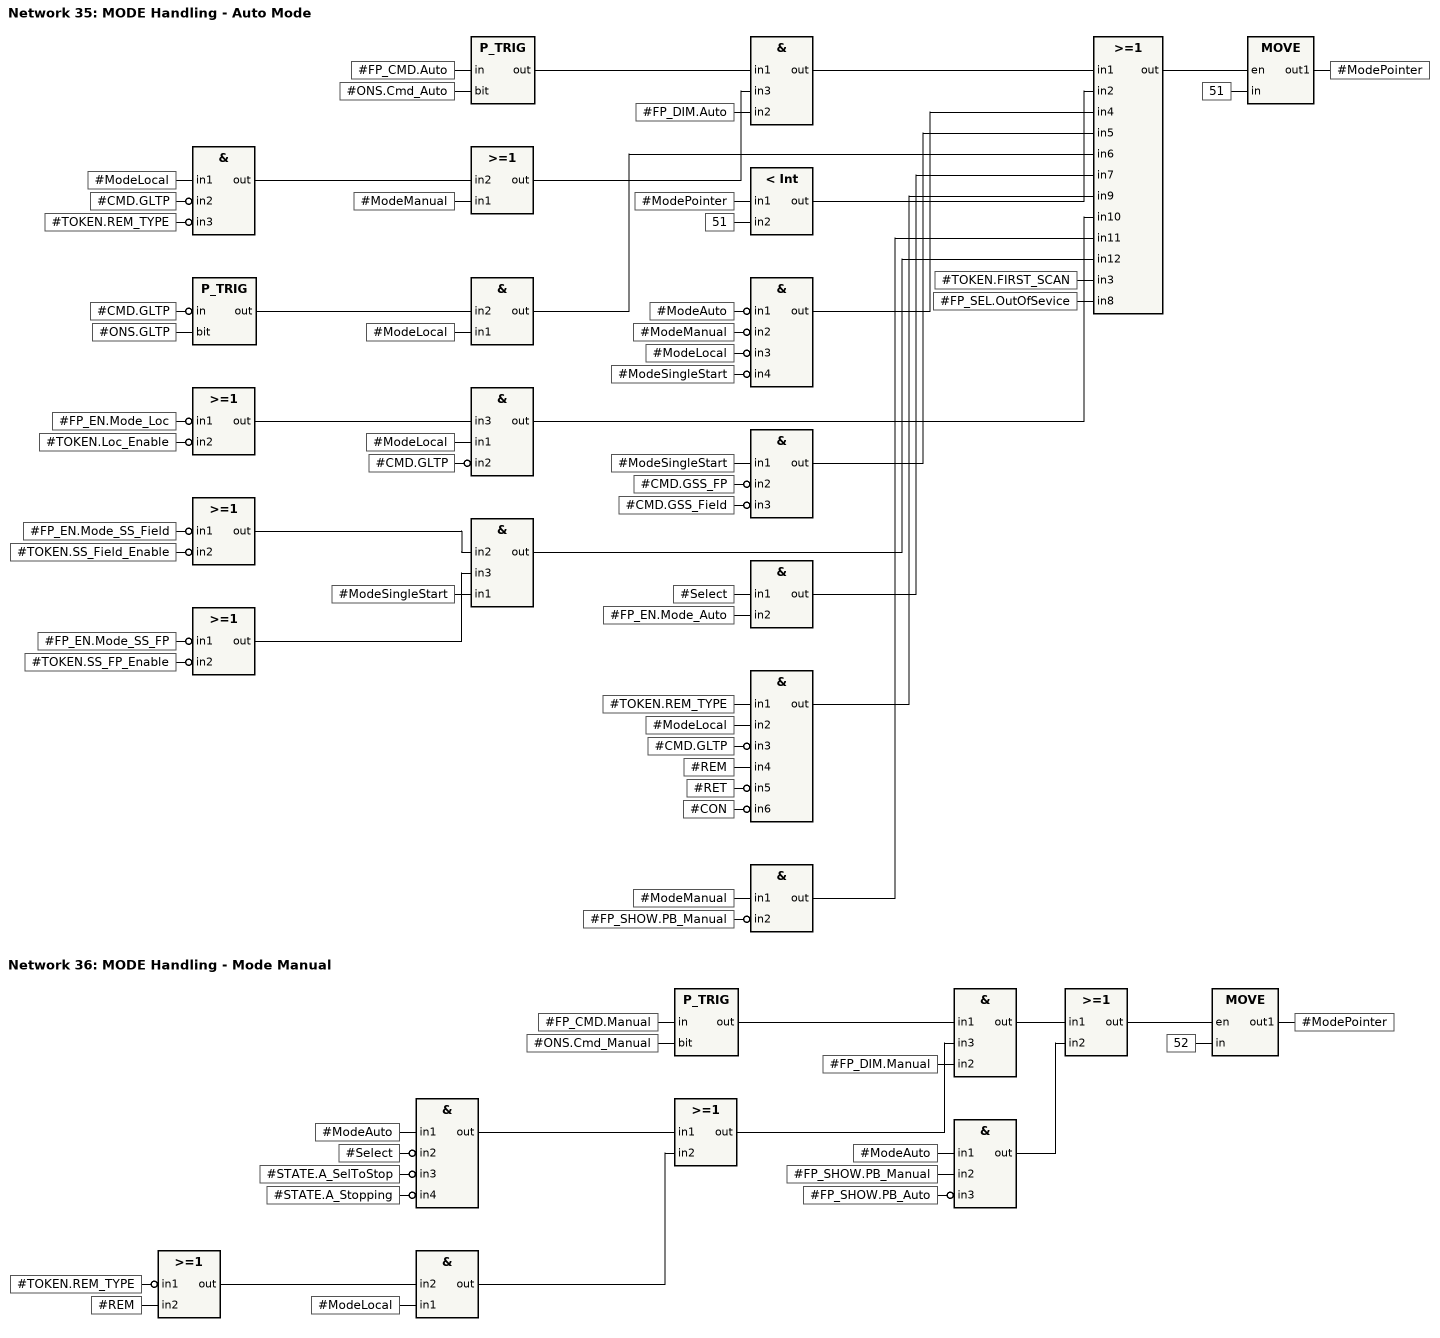
   #_w1 := #FP_CMD.Auto AND NOT #ONS.Cmd_Auto;   // rising edge
   #ONS.Cmd_Auto := #FP_CMD.Auto;
   #_w2 := NOT #CMD.GLTP AND NOT #ONS.GLTP;   // rising edge
   #ONS.GLTP := NOT #CMD.GLTP;
   IF (#_w1 AND ((#ModeLocal AND NOT #CMD.GLTP AND NOT #TOKEN.REM_TYPE) OR #ModeManual) AND #FP_DIM.Auto) OR (#ModePointer < 51) OR (NOT #ModeAuto AND NOT #ModeManual AND NOT #ModeLocal AND NOT #ModeSingleStart) OR (#ModeSingleStart AND NOT #CMD.GSS_FP AND NOT #CMD.GSS_Field) OR (#_w2 AND #ModeLocal) OR (#Select AND #FP_EN.Mode_Auto) OR (#TOKEN.REM_TYPE AND #ModeLocal AND NOT #CMD.GLTP AND #REM AND NOT #RET AND NOT #CON) OR ((NOT #FP_EN.Mode_Loc OR NOT #TOKEN.Loc_Enable) AND #ModeLocal AND NOT #CMD.GLTP) OR (#ModeManual AND NOT #FP_SHOW.PB_Manual) OR ((NOT #FP_EN.Mode_SS_Field OR NOT #TOKEN.SS_Field_Enable) AND (NOT #FP_EN.Mode_SS_FP OR NOT #TOKEN.SS_FP_Enable) AND #ModeSingleStart) OR #TOKEN.FIRST_SCAN OR #FP_SEL.OutOfSevice THEN
       #ModePointer := 51;
   END_IF;
END_REGION

REGION Network 36: MODE Handling - Mode Manual
   #_w1 := #FP_CMD.Manual AND NOT #ONS.Cmd_Manual;   // rising edge
   #ONS.Cmd_Manual := #FP_CMD.Manual;
   IF (#_w1 AND ((#ModeAuto AND NOT #Select AND NOT #STATE.A_SelToStop AND NOT #STATE.A_Stopping) OR ((NOT #TOKEN.REM_TYPE OR #REM) AND #ModeLocal)) AND #FP_DIM.Manual) OR (#ModeAuto AND #FP_SHOW.PB_Manual AND NOT #FP_SHOW.PB_Auto) THEN
       #ModePointer := 52;
   END_IF;
END_REGION

REGION Network 37: MODE Handling - Mode Single Start
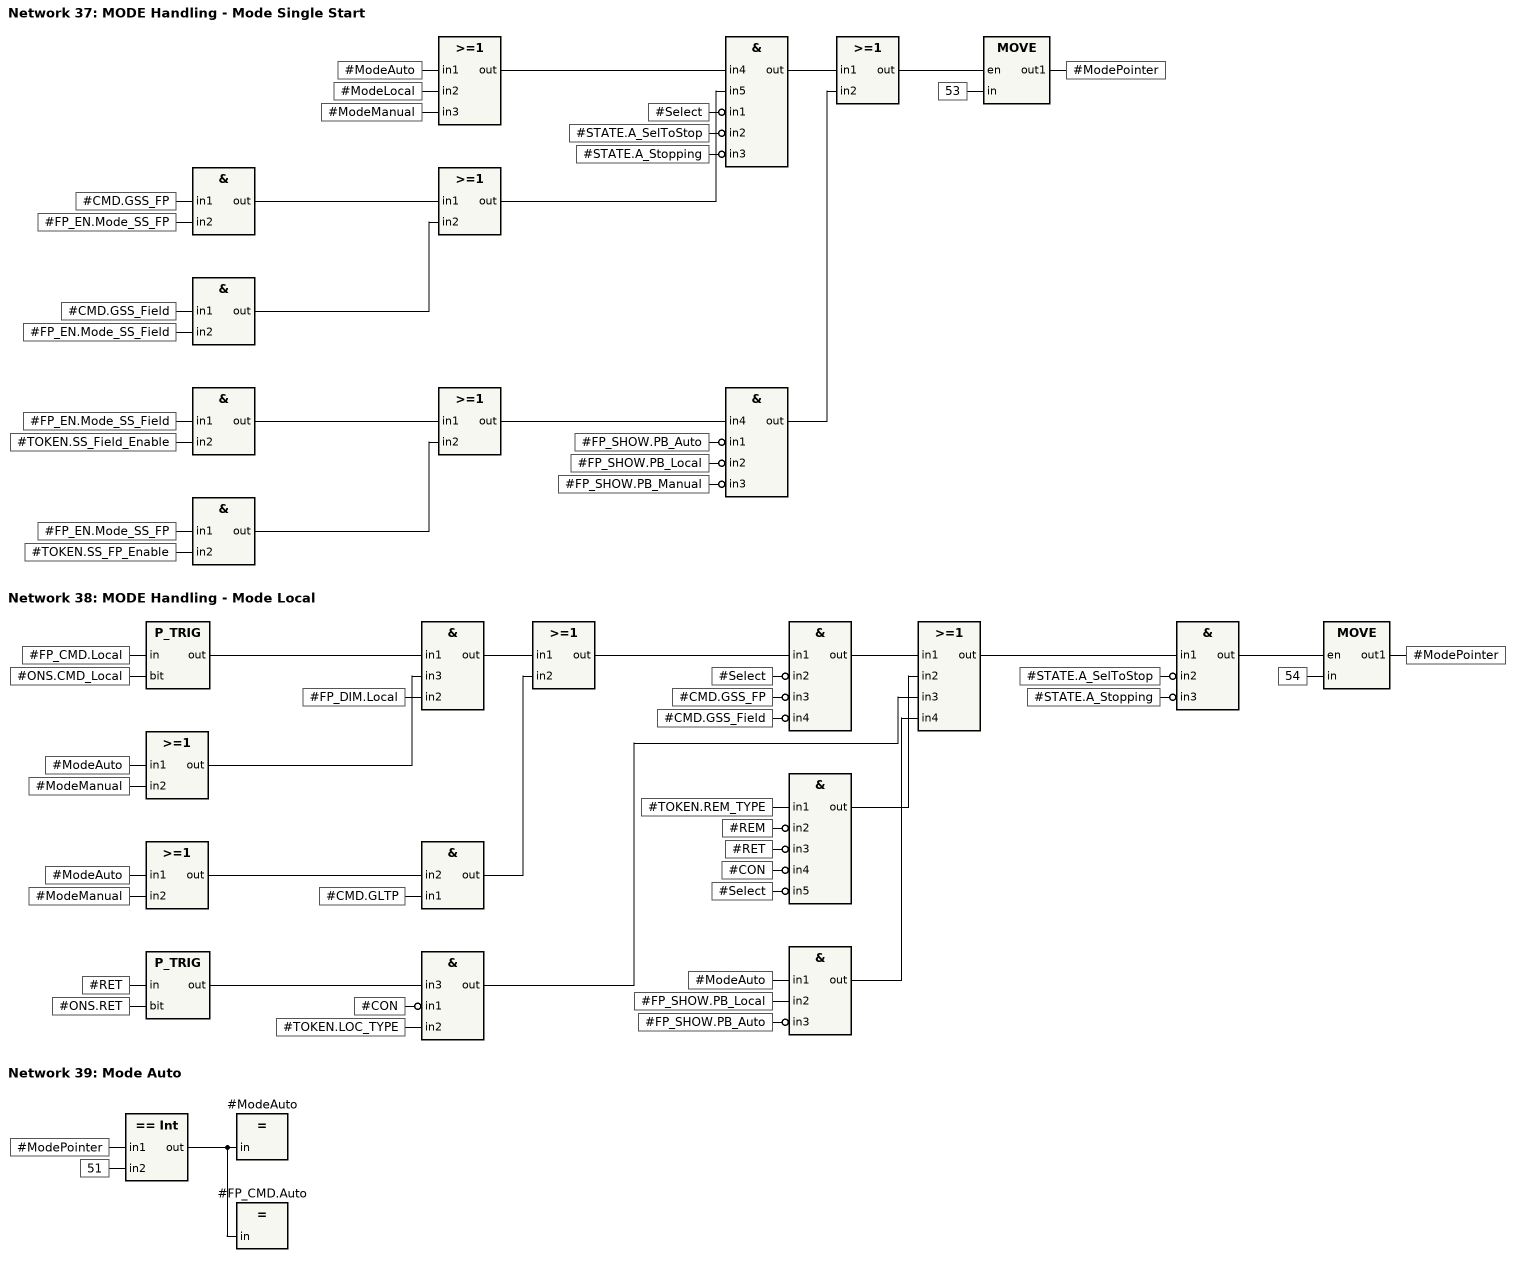
   IF ((#ModeAuto OR #ModeLocal OR #ModeManual) AND ((#CMD.GSS_FP AND #FP_EN.Mode_SS_FP) OR (#CMD.GSS_Field AND #FP_EN.Mode_SS_Field)) AND NOT #Select AND NOT #STATE.A_SelToStop AND NOT #STATE.A_Stopping) OR (((#FP_EN.Mode_SS_Field AND #TOKEN.SS_Field_Enable) OR (#FP_EN.Mode_SS_FP AND #TOKEN.SS_FP_Enable)) AND NOT #FP_SHOW.PB_Auto AND NOT #FP_SHOW.PB_Local AND NOT #FP_SHOW.PB_Manual) THEN
       #ModePointer := 53;
   END_IF;
END_REGION

REGION Network 38: MODE Handling - Mode Local
   #_w1 := #FP_CMD.Local AND NOT #ONS.CMD_Local;   // rising edge
   #ONS.CMD_Local := #FP_CMD.Local;
   #_w2 := #RET AND NOT #ONS.RET;   // rising edge
   #ONS.RET := #RET;
   IF ((((#_w1 AND (#ModeAuto OR #ModeManual) AND #FP_DIM.Local) OR ((#ModeAuto OR #ModeManual) AND #CMD.GLTP)) AND NOT #Select AND NOT #CMD.GSS_FP AND NOT #CMD.GSS_Field) OR (#TOKEN.REM_TYPE AND NOT #REM AND NOT #RET AND NOT #CON AND NOT #Select) OR (#_w2 AND NOT #CON AND #TOKEN.LOC_TYPE) OR (#ModeAuto AND #FP_SHOW.PB_Local AND NOT #FP_SHOW.PB_Auto)) AND NOT #STATE.A_SelToStop AND NOT #STATE.A_Stopping THEN
       #ModePointer := 54;
   END_IF;
END_REGION

REGION Network 39: Mode Auto
   #ModeAuto := #ModePointer = 51;
   #FP_CMD.Auto := #ModeAuto;
END_REGION

REGION Network 40: Mode Manual
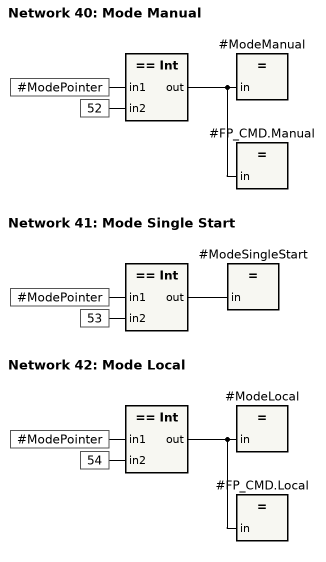
   #ModeManual := #ModePointer = 52;
   #FP_CMD.Manual := #ModeManual;
END_REGION

REGION Network 41: Mode Single Start
   #ModeSingleStart := #ModePointer = 53;
END_REGION

REGION Network 42: Mode Local
   #ModeLocal := #ModePointer = 54;
   #FP_CMD.Local := #ModeLocal;
END_REGION

REGION Network 43: FACEPLATE COMMANDS (Pulse Type)
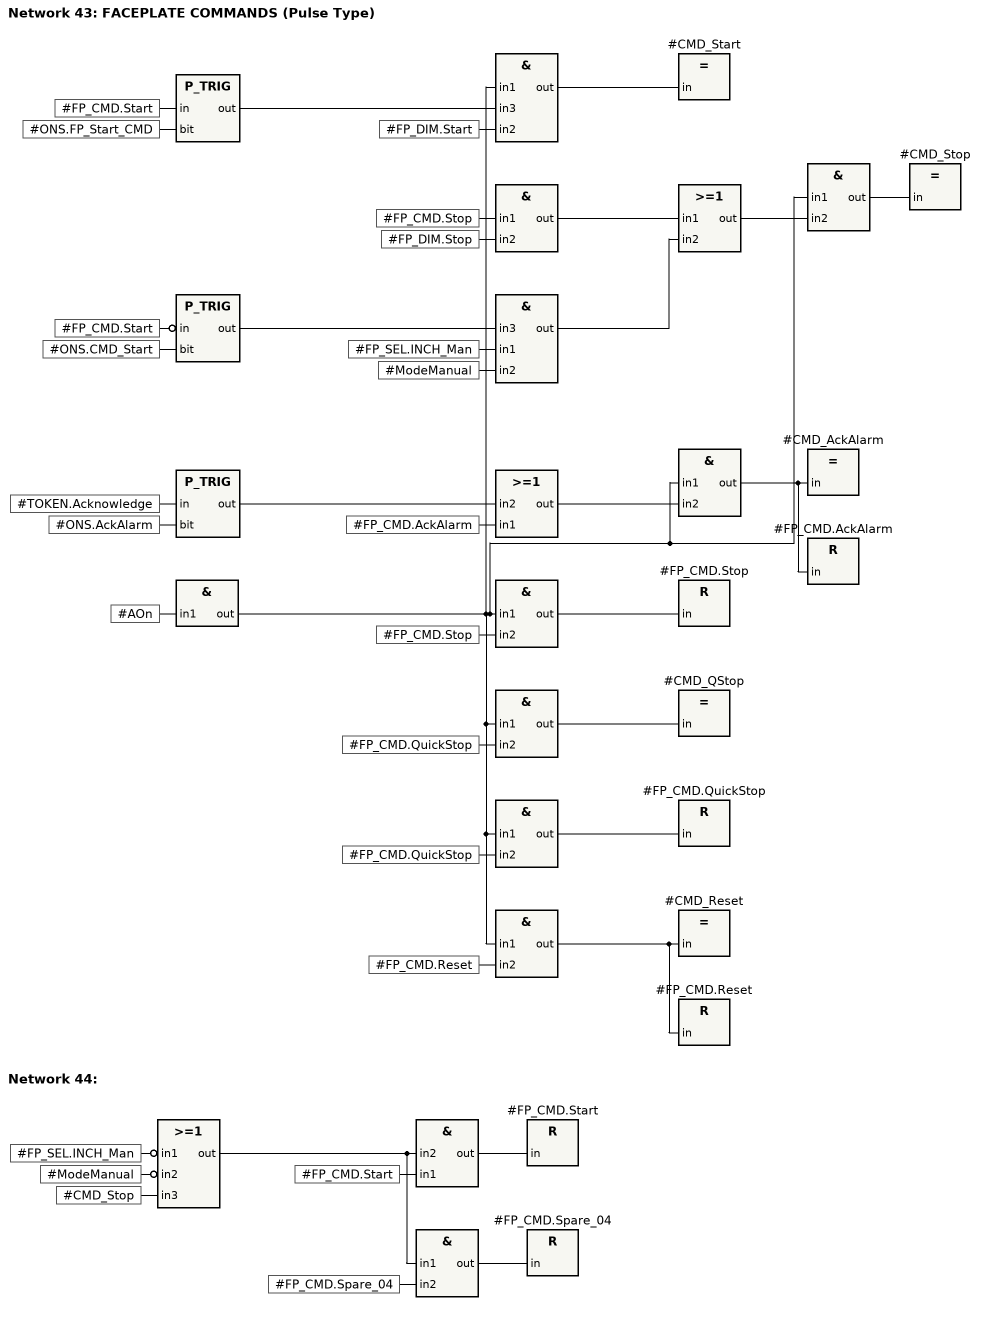
   #_w1 := #FP_CMD.Start AND NOT #ONS.FP_Start_CMD;   // rising edge
   #ONS.FP_Start_CMD := #FP_CMD.Start;
   #CMD_Start := #AOn AND #_w1 AND #FP_DIM.Start;
   #_w2 := NOT #FP_CMD.Start AND NOT #ONS.CMD_Start;   // rising edge
   #ONS.CMD_Start := NOT #FP_CMD.Start;
   #CMD_Stop := #AOn AND ((#FP_CMD.Stop AND #FP_DIM.Stop) OR (#_w2 AND #FP_SEL.INCH_Man AND #ModeManual));
   IF #AOn AND #FP_CMD.Stop THEN #FP_CMD.Stop := FALSE; END_IF;
   #CMD_QStop := #AOn AND #FP_CMD.QuickStop;
   IF #AOn AND #FP_CMD.QuickStop THEN #FP_CMD.QuickStop := FALSE; END_IF;
   #CMD_Reset := #AOn AND #FP_CMD.Reset;
   IF #CMD_Reset THEN #FP_CMD.Reset := FALSE; END_IF;
   #_w3 := #TOKEN.Acknowledge AND NOT #ONS.AckAlarm;   // rising edge
   #ONS.AckAlarm := #TOKEN.Acknowledge;
   #CMD_AckAlarm := #AOn AND (#_w3 OR #FP_CMD.AckAlarm);
   IF #CMD_AckAlarm THEN #FP_CMD.AckAlarm := FALSE; END_IF;
END_REGION

REGION Network 44
   #_w1 := NOT #FP_SEL.INCH_Man OR NOT #ModeManual OR #CMD_Stop;
   IF #_w1 AND #FP_CMD.Start THEN #FP_CMD.Start := FALSE; END_IF;
   IF #_w1 AND #FP_CMD.Spare_04 THEN #FP_CMD.Spare_04 := FALSE; END_IF;
END_REGION

REGION Network 45: ALARM SUPPRESSION
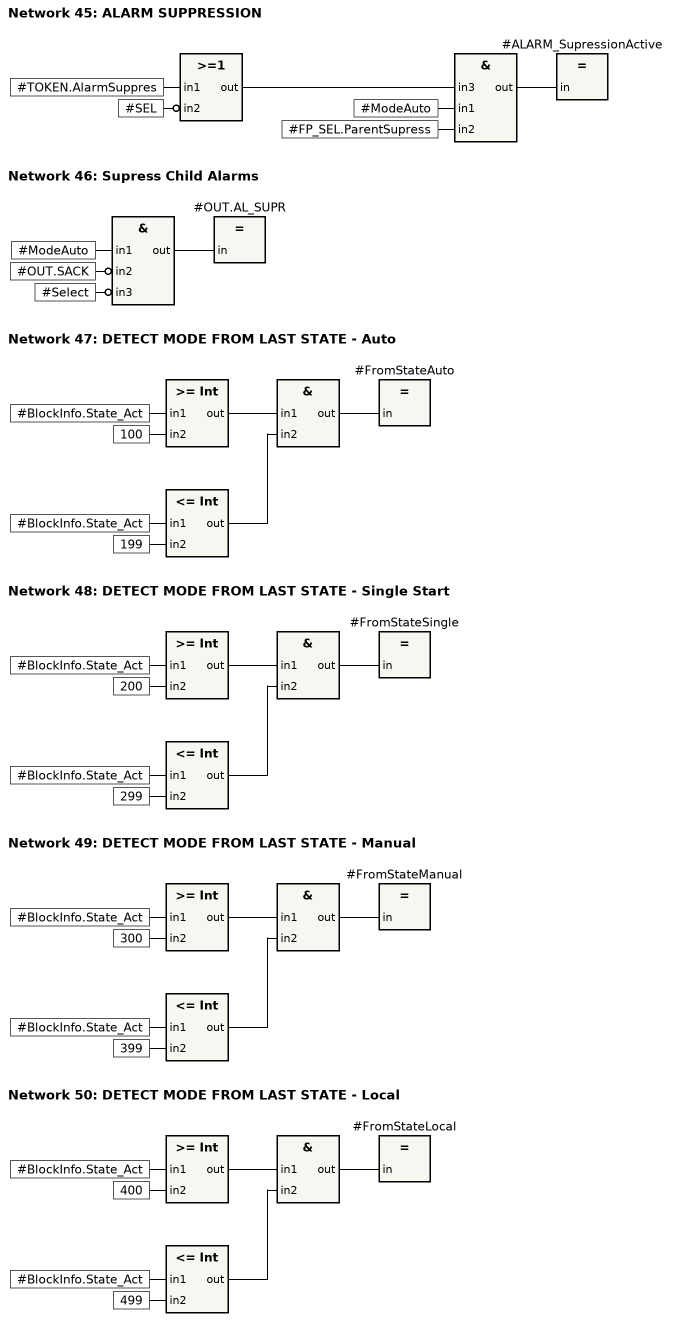
   #ALARM_SupressionActive := (#TOKEN.AlarmSuppres OR NOT #SEL) AND #ModeAuto AND #FP_SEL.ParentSupress;
END_REGION

REGION Network 46: Supress Child Alarms
   #OUT.AL_SUPR := #ModeAuto AND NOT #OUT.SACK AND NOT #Select;
END_REGION

REGION Network 47: DETECT MODE FROM LAST STATE - Auto
   #FromStateAuto := (#BlockInfo.State_Act >= 100) AND (#BlockInfo.State_Act <= 199);
END_REGION

REGION Network 48: DETECT MODE FROM LAST STATE - Single Start
   #FromStateSingle := (#BlockInfo.State_Act >= 200) AND (#BlockInfo.State_Act <= 299);
END_REGION

REGION Network 49: DETECT MODE FROM LAST STATE - Manual
   #FromStateManual := (#BlockInfo.State_Act >= 300) AND (#BlockInfo.State_Act <= 399);
END_REGION

REGION Network 50: DETECT MODE FROM LAST STATE - Local
   #FromStateLocal := (#BlockInfo.State_Act >= 400) AND (#BlockInfo.State_Act <= 499);
END_REGION

REGION Network 51: DETECT MODE FROM LAST STATE - Stop
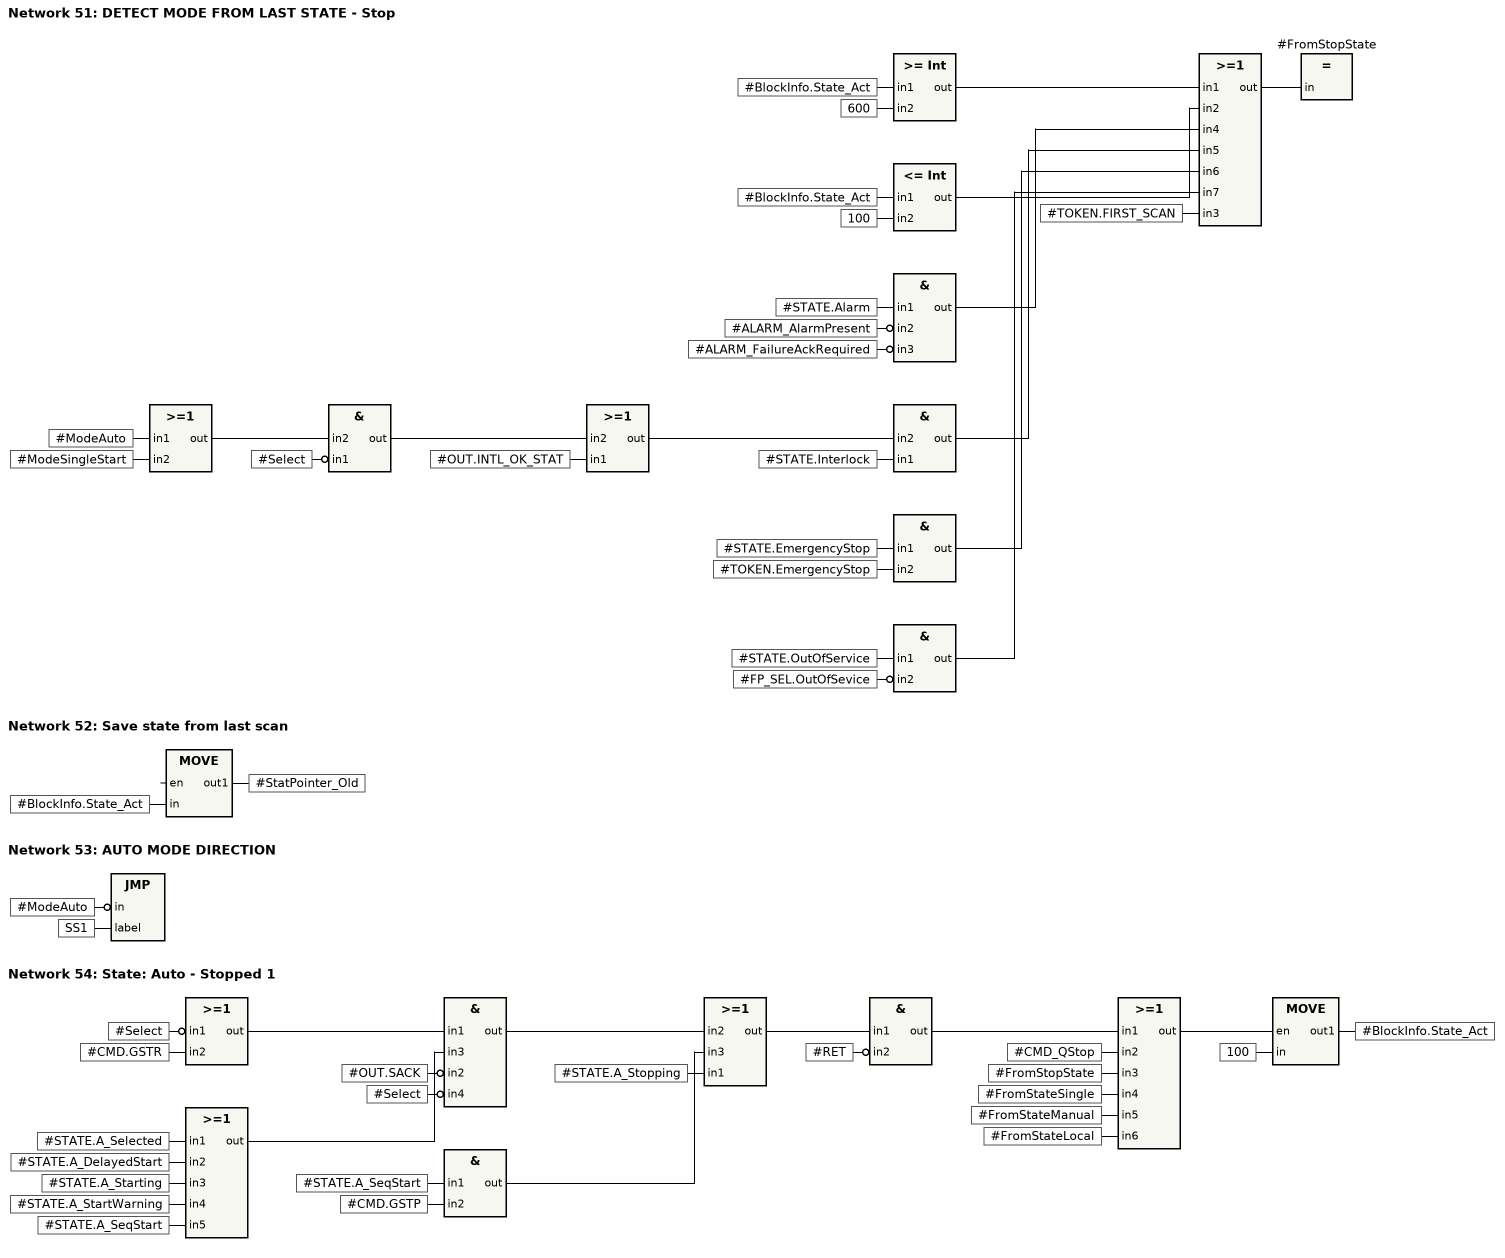
   #FromStopState := (#BlockInfo.State_Act >= 600) OR (#BlockInfo.State_Act <= 100) OR (#STATE.Alarm AND NOT #ALARM_AlarmPresent AND NOT #ALARM_FailureAckRequired) OR ((((#ModeAuto OR #ModeSingleStart) AND NOT #Select) OR #OUT.INTL_OK_STAT) AND #STATE.Interlock) OR (#STATE.EmergencyStop AND #TOKEN.EmergencyStop) OR (#STATE.OutOfService AND NOT #FP_SEL.OutOfSevice) OR #TOKEN.FIRST_SCAN;
END_REGION

REGION Network 52: Save state from last scan
   #StatPointer_Old := #BlockInfo.State_Act;
END_REGION

REGION Network 53: AUTO MODE DIRECTION
   IF NOT #ModeAuto THEN GOTO SS1; END_IF;
END_REGION

REGION Network 54: State: Auto - Stopped 1
   IF ((((NOT #Select OR #CMD.GSTR) AND (#STATE.A_Selected OR #STATE.A_DelayedStart OR #STATE.A_Starting OR #STATE.A_StartWarning OR #STATE.A_SeqStart) AND NOT #OUT.SACK AND NOT #Select) OR (#STATE.A_SeqStart AND #CMD.GSTP) OR #STATE.A_Stopping) AND NOT #RET) OR #CMD_QStop OR #FromStopState OR #FromStateSingle OR #FromStateManual OR #FromStateLocal THEN
       #BlockInfo.State_Act := 100;
   END_IF;
END_REGION

REGION Network 55: State: Auto - Selected 1
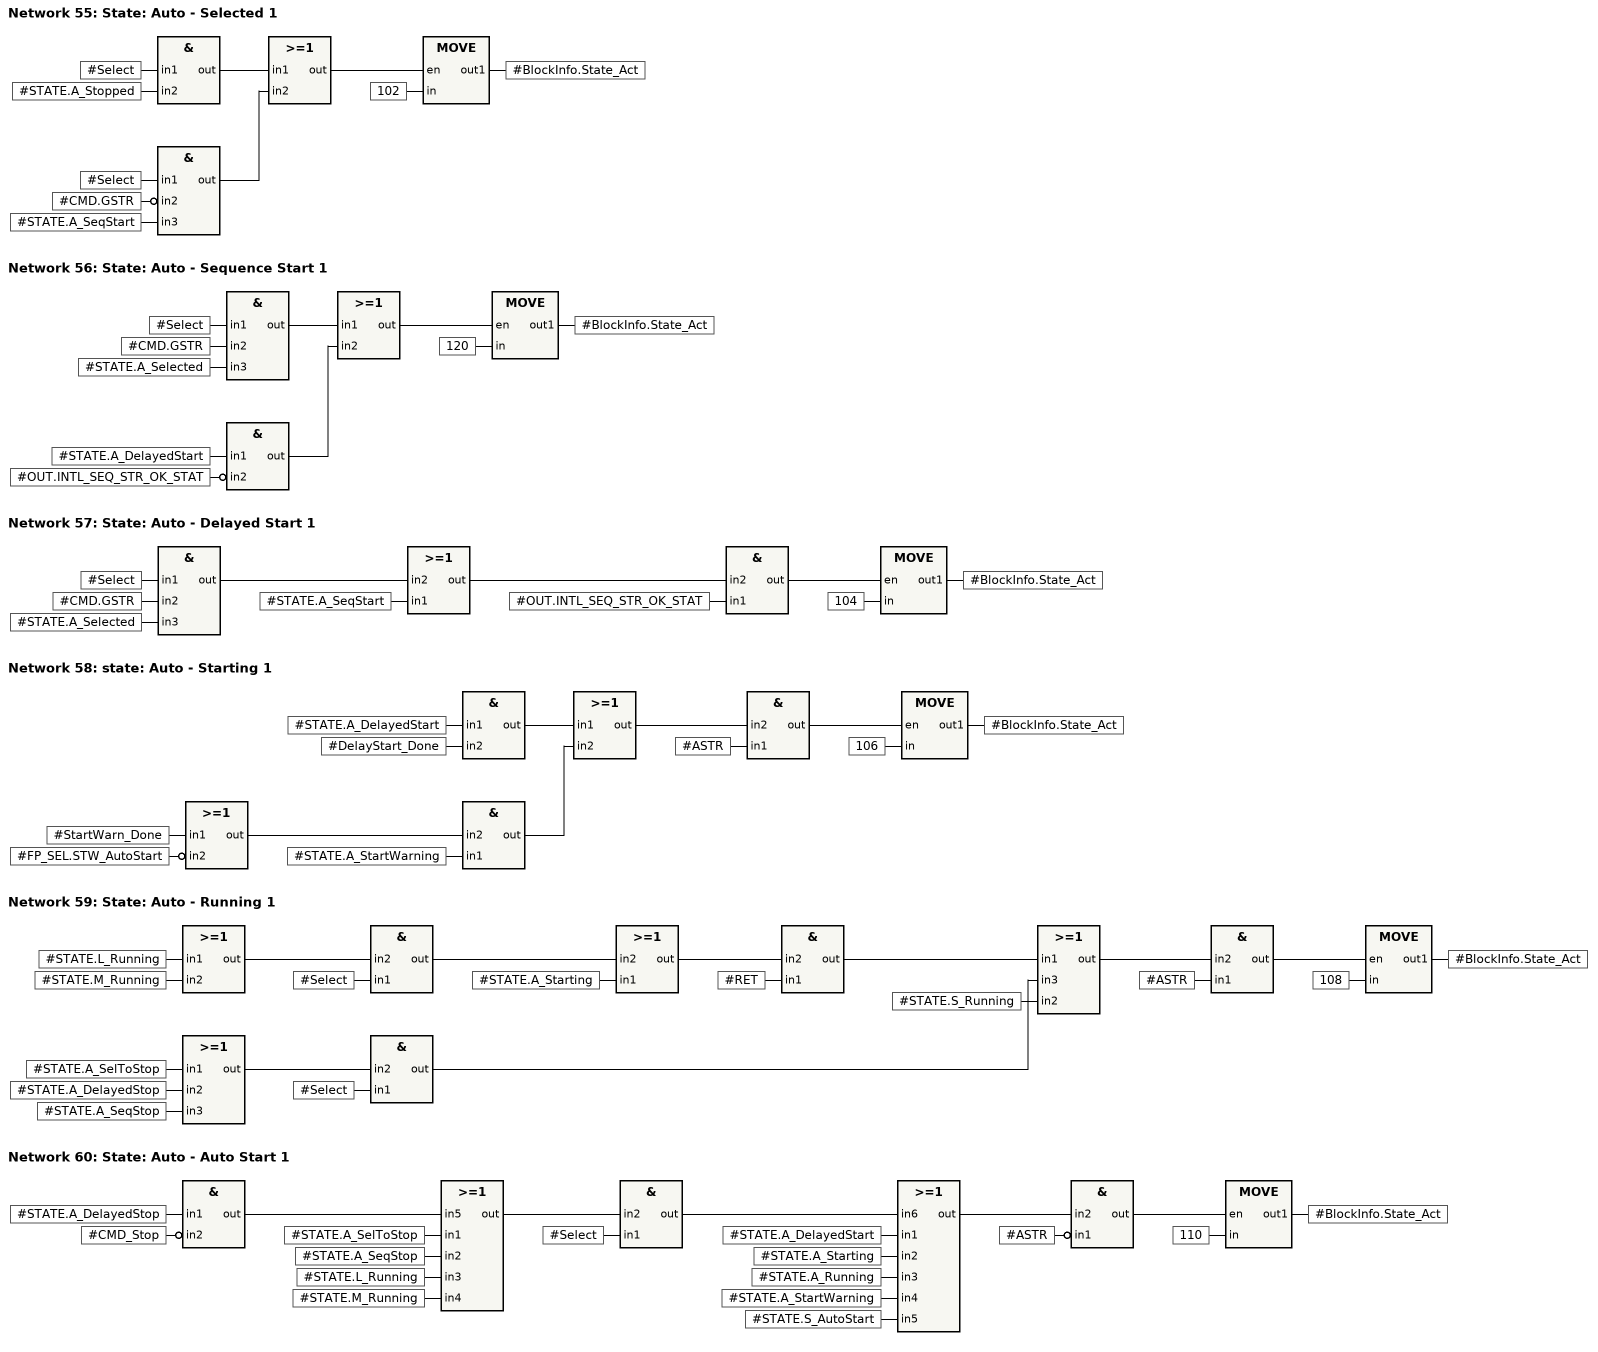
   IF (#Select AND #STATE.A_Stopped) OR (#Select AND NOT #CMD.GSTR AND #STATE.A_SeqStart) THEN
       #BlockInfo.State_Act := 102;
   END_IF;
END_REGION

REGION Network 56: State: Auto - Sequence Start 1
   IF (#Select AND #CMD.GSTR AND #STATE.A_Selected) OR (#STATE.A_DelayedStart AND NOT #OUT.INTL_SEQ_STR_OK_STAT) THEN
       #BlockInfo.State_Act := 120;
   END_IF;
END_REGION

REGION Network 57: State: Auto - Delayed Start 1
   IF ((#Select AND #CMD.GSTR AND #STATE.A_Selected) OR #STATE.A_SeqStart) AND #OUT.INTL_SEQ_STR_OK_STAT THEN
       #BlockInfo.State_Act := 104;
   END_IF;
END_REGION

REGION Network 58: state: Auto - Starting 1
   IF ((#STATE.A_DelayedStart AND #DelayStart_Done) OR ((#StartWarn_Done OR NOT #FP_SEL.STW_AutoStart) AND #STATE.A_StartWarning)) AND #ASTR THEN
       #BlockInfo.State_Act := 106;
   END_IF;
END_REGION

REGION Network 59: State: Auto - Running 1
   IF (((((#STATE.L_Running OR #STATE.M_Running) AND #Select) OR #STATE.A_Starting) AND #RET) OR ((#STATE.A_SelToStop OR #STATE.A_DelayedStop OR #STATE.A_SeqStop) AND #Select) OR #STATE.S_Running) AND #ASTR THEN
       #BlockInfo.State_Act := 108;
   END_IF;
END_REGION

REGION Network 60: State: Auto - Auto Start 1
   IF ((((#STATE.A_DelayedStop AND NOT #CMD_Stop) OR #STATE.A_SelToStop OR #STATE.A_SeqStop OR #STATE.L_Running OR #STATE.M_Running) AND #Select) OR #STATE.A_DelayedStart OR #STATE.A_Starting OR #STATE.A_Running OR #STATE.A_StartWarning OR #STATE.S_AutoStart) AND NOT #ASTR THEN
       #BlockInfo.State_Act := 110;
   END_IF;
END_REGION

REGION Network 61: State: Auto - Selected to Stop 1
   // Build 003 - 11 Jul 2019 (EXTBOB) : GSEL added to A_SeqStop with GSTP condition to move to Selected to Stop state from Seq stop state if group stop timer completes
